Yaskawa INFORM job: A_ROOF_SIDE_0617_2_PAINT_8.JBI

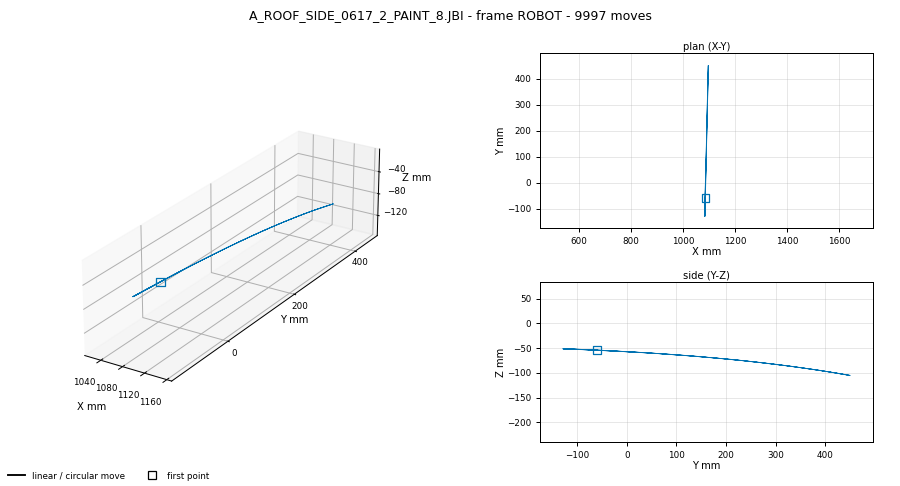
[picture p0: tool path of A_ROOF_SIDE_0617_2_PAINT_8.JBI in frame ROBOT, 9997 of 9997 moves have a stored position in this frame; points joined in program order, loops and branches not executed]
/JOB
//NAME A_ROOF_SIDE_0617_2_PAINT8
//POS
///NPOS 9997,0,0,0,0,0
///TOOL 1
///USER 0
///POSTYPE ROBOT
///RECTAN
///RCONF 1,0,0,0,0,0,0,0,0,0,0,0,0,0,0,0,0,0,0,0,0,0,0,0
C00000=1085.581,-59.825,-53.867,174.286,17.983,152.948
C00001=1085.575,-60.075,-53.857,174.285,17.982,152.948
C00002=1085.569,-60.325,-53.845,174.283,17.980,152.948
C00003=1085.563,-60.574,-53.833,174.282,17.979,152.948
C00004=1085.557,-60.824,-53.822,174.280,17.978,152.948
C00005=1085.551,-61.074,-53.811,174.279,17.976,152.948
C00006=1085.545,-61.323,-53.799,174.277,17.974,152.948
C00007=1085.540,-61.573,-53.788,174.276,17.973,152.948
C00008=1085.534,-61.823,-53.777,174.274,17.972,152.948
C00009=1085.527,-62.072,-53.765,174.273,17.970,152.948
C00010=1085.522,-62.322,-53.754,174.272,17.969,152.948
C00011=1085.515,-62.572,-53.743,174.270,17.968,152.948
C00012=1085.509,-62.821,-53.731,174.269,17.966,152.948
C00013=1085.504,-63.071,-53.719,174.267,17.965,152.948
C00014=1085.498,-63.321,-53.708,174.265,17.963,152.948
C00015=1085.491,-63.571,-53.697,174.264,17.962,152.948
C00016=1085.485,-63.820,-53.685,174.263,17.960,152.948
C00017=1085.480,-64.069,-53.675,174.261,17.959,152.948
C00018=1085.473,-64.320,-53.663,174.260,17.958,152.948
C00019=1085.468,-64.569,-53.651,174.258,17.956,152.948
C00020=1085.461,-64.842,-53.640,174.257,17.955,152.948
C00021=1085.455,-65.116,-53.627,174.254,17.953,152.948
C00022=1085.448,-65.389,-53.615,174.253,17.951,152.948
C00023=1085.442,-65.662,-53.602,174.252,17.950,152.948
C00024=1085.436,-65.912,-53.591,174.250,17.948,152.948
C00025=1085.430,-66.162,-53.580,174.248,17.947,152.948
C00026=1085.424,-66.411,-53.569,174.247,17.946,152.948
C00027=1085.418,-66.661,-53.557,174.246,17.944,152.948
C00028=1085.412,-66.911,-53.546,174.244,17.943,152.948
C00029=1085.407,-67.160,-53.535,174.243,17.942,152.948
C00030=1085.400,-67.410,-53.524,174.241,17.940,152.948
C00031=1085.394,-67.660,-53.513,174.240,17.939,152.948
C00032=1085.389,-67.909,-53.502,174.238,17.937,152.948
C00033=1085.382,-68.159,-53.490,174.237,17.936,152.948
C00034=1085.376,-68.409,-53.479,174.235,17.935,152.948
C00035=1085.371,-68.658,-53.468,174.234,17.933,152.948
C00036=1085.365,-68.909,-53.456,174.232,17.932,152.948
C00037=1085.359,-69.158,-53.445,174.231,17.931,152.948
C00038=1085.354,-69.407,-53.435,174.229,17.929,152.948
C00039=1085.347,-69.658,-53.423,174.228,17.928,152.948
C00040=1085.341,-69.907,-53.412,174.226,17.926,152.948
C00041=1085.336,-70.157,-53.402,174.225,17.925,152.948
C00042=1085.329,-70.406,-53.390,174.223,17.924,152.948
C00043=1085.323,-70.656,-53.379,174.222,17.922,152.948
C00044=1085.318,-70.905,-53.368,174.220,17.921,152.948
C00045=1085.311,-71.155,-53.357,174.219,17.920,152.948
C00046=1085.306,-71.405,-53.346,174.217,17.918,152.948
C00047=1085.300,-71.655,-53.334,174.216,17.917,152.948
C00048=1085.294,-71.905,-53.323,174.214,17.915,152.948
C00049=1085.288,-72.154,-53.312,174.213,17.914,152.948
C00050=1085.283,-72.404,-53.301,174.211,17.913,152.949
C00051=1085.277,-72.653,-53.290,174.210,17.911,152.948
C00052=1085.271,-72.904,-53.279,174.208,17.910,152.948
C00053=1085.265,-73.153,-53.268,174.207,17.909,152.949
C00054=1085.259,-73.403,-53.257,174.205,17.907,152.949
C00055=1085.253,-73.652,-53.246,174.204,17.906,152.949
C00056=1085.247,-73.902,-53.235,174.202,17.904,152.949
C00057=1085.241,-74.152,-53.224,174.201,17.903,152.949
C00058=1085.236,-74.401,-53.213,174.199,17.902,152.949
C00059=1085.229,-74.651,-53.202,174.198,17.900,152.949
C00060=1085.223,-74.901,-53.191,174.196,17.899,152.949
C00061=1085.218,-75.150,-53.180,174.195,17.898,152.949
C00062=1085.211,-75.400,-53.170,174.193,17.896,152.949
C00063=1085.205,-75.650,-53.159,174.192,17.895,152.949
C00064=1085.199,-75.899,-53.148,174.190,17.894,152.949
C00065=1085.193,-76.149,-53.137,174.188,17.893,152.949
C00066=1085.187,-76.399,-53.126,174.187,17.891,152.949
C00067=1085.181,-76.648,-53.115,174.185,17.890,152.949
C00068=1085.176,-76.898,-53.104,174.184,17.889,152.949
C00069=1085.169,-77.148,-53.094,174.182,17.888,152.949
C00070=1085.163,-77.398,-53.083,174.181,17.886,152.949
C00071=1085.157,-77.647,-53.073,174.179,17.885,152.949
C00072=1085.152,-77.897,-53.062,174.178,17.883,152.949
C00073=1085.145,-78.147,-53.050,174.176,17.882,152.949
C00074=1085.140,-78.397,-53.040,174.175,17.881,152.949
C00075=1085.133,-78.646,-53.029,174.174,17.880,152.949
C00076=1085.127,-78.895,-53.018,174.172,17.879,152.949
C00077=1085.121,-79.145,-53.007,174.171,17.878,152.949
C00078=1085.115,-79.395,-52.996,174.169,17.876,152.949
C00079=1085.110,-79.645,-52.986,174.168,17.875,152.949
C00080=1085.104,-79.894,-52.975,174.166,17.874,152.950
C00081=1085.097,-80.144,-52.965,174.165,17.872,152.950
C00082=1085.091,-80.394,-52.954,174.163,17.871,152.950
C00083=1085.086,-80.643,-52.943,174.162,17.870,152.950
C00084=1085.079,-80.920,-52.931,174.160,17.869,152.950
C00085=1085.072,-81.195,-52.919,174.158,17.868,152.950
C00086=1085.065,-81.470,-52.907,174.157,17.866,152.950
C00087=1085.059,-81.746,-52.896,174.154,17.865,152.950
C00088=1085.052,-81.995,-52.886,174.153,17.863,152.950
C00089=1085.046,-82.245,-52.874,174.152,17.862,152.950
C00090=1085.040,-82.495,-52.864,174.150,17.861,152.950
C00091=1085.034,-82.744,-52.854,174.149,17.860,152.950
C00092=1085.028,-82.994,-52.843,174.147,17.859,152.950
C00093=1085.022,-83.244,-52.832,174.146,17.858,152.950
C00094=1085.015,-83.493,-52.822,174.144,17.857,152.950
C00095=1085.010,-83.743,-52.811,174.143,17.855,152.950
C00096=1085.003,-83.993,-52.801,174.141,17.854,152.950
C00097=1084.997,-84.243,-52.790,174.139,17.853,152.951
C00098=1084.991,-84.492,-52.779,174.138,17.851,152.951
C00099=1084.985,-84.742,-52.769,174.136,17.850,152.951
C00100=1084.979,-84.992,-52.759,174.135,17.849,152.951
C00101=1084.972,-85.241,-52.748,174.133,17.848,152.951
C00102=1084.967,-85.492,-52.738,174.132,17.847,152.951
C00103=1084.961,-85.741,-52.727,174.131,17.846,152.951
C00104=1084.955,-85.990,-52.717,174.129,17.845,152.951
C00105=1084.949,-86.240,-52.706,174.128,17.844,152.951
C00106=1084.943,-86.491,-52.695,174.126,17.842,152.951
C00107=1084.936,-86.740,-52.685,174.124,17.841,152.951
C00108=1084.931,-86.990,-52.675,174.123,17.840,152.951
C00109=1084.924,-87.239,-52.665,174.121,17.839,152.951
C00110=1084.919,-87.488,-52.654,174.120,17.838,152.951
C00111=1084.912,-87.739,-52.644,174.118,17.836,152.951
C00112=1084.906,-87.988,-52.633,174.117,17.835,152.952
C00113=1084.900,-88.238,-52.622,174.115,17.834,152.952
C00114=1084.894,-88.488,-52.612,174.114,17.834,152.952
C00115=1084.889,-88.737,-52.602,174.113,17.832,152.952
C00116=1084.882,-88.986,-52.591,174.111,17.831,152.952
C00117=1084.876,-89.237,-52.581,174.109,17.830,152.952
C00118=1084.870,-89.486,-52.570,174.108,17.829,152.952
C00119=1084.864,-89.737,-52.560,174.106,17.827,152.952
C00120=1084.858,-89.986,-52.549,174.105,17.826,152.952
C00121=1084.852,-90.235,-52.539,174.103,17.825,152.952
C00122=1084.847,-90.485,-52.529,174.101,17.824,152.952
C00123=1084.840,-90.734,-52.519,174.101,17.823,152.952
C00124=1084.834,-90.985,-52.508,174.099,17.822,152.952
C00125=1084.828,-91.234,-52.498,174.097,17.821,152.952
C00126=1084.822,-91.485,-52.488,174.096,17.820,152.953
C00127=1084.816,-91.734,-52.477,174.094,17.819,152.953
C00128=1084.810,-91.984,-52.467,174.093,17.817,152.953
C00129=1084.804,-92.233,-52.457,174.091,17.816,152.953
C00130=1084.798,-92.483,-52.446,174.089,17.815,152.953
C00131=1084.793,-92.733,-52.436,174.088,17.814,152.953
C00132=1084.786,-92.982,-52.426,174.087,17.813,152.953
C00133=1084.780,-93.233,-52.415,174.085,17.812,152.953
C00134=1084.774,-93.482,-52.405,174.084,17.811,152.953
C00135=1084.768,-93.732,-52.395,174.082,17.810,152.953
C00136=1084.762,-93.981,-52.384,174.080,17.809,152.953
C00137=1084.756,-94.231,-52.374,174.079,17.807,152.953
C00138=1084.750,-94.480,-52.364,174.077,17.806,152.953
C00139=1084.744,-94.731,-52.354,174.076,17.805,152.954
C00140=1084.738,-94.980,-52.344,174.074,17.804,152.954
C00141=1084.732,-95.230,-52.333,174.073,17.804,152.954
C00142=1084.726,-95.480,-52.324,174.072,17.803,152.954
C00143=1084.720,-95.729,-52.313,174.070,17.801,152.954
C00144=1084.714,-95.979,-52.303,174.068,17.800,152.954
C00145=1084.709,-96.228,-52.292,174.067,17.799,152.954
C00146=1084.702,-96.478,-52.283,174.065,17.798,152.954
C00147=1084.697,-96.728,-52.273,174.063,17.797,152.954
C00148=1084.688,-97.066,-52.259,174.062,17.796,152.954
C00149=1084.680,-97.404,-52.245,174.060,17.794,152.954
C00150=1084.672,-97.741,-52.231,174.058,17.793,152.954
C00151=1084.664,-98.079,-52.218,174.055,17.791,152.955
C00152=1084.658,-98.328,-52.207,174.054,17.790,152.955
C00153=1084.652,-98.578,-52.198,174.053,17.789,152.955
C00154=1084.645,-98.828,-52.188,174.051,17.788,152.955
C00155=1084.640,-99.077,-52.177,174.050,17.787,152.955
C00156=1084.633,-99.328,-52.167,174.048,17.786,152.955
C00157=1084.627,-99.577,-52.158,174.046,17.785,152.955
C00158=1084.621,-99.827,-52.147,174.045,17.784,152.955
C00159=1084.615,-100.077,-52.137,174.044,17.784,152.955
C00160=1084.609,-100.326,-52.128,174.042,17.783,152.956
C00161=1084.603,-100.576,-52.117,174.040,17.782,152.956
C00162=1084.597,-100.826,-52.107,174.039,17.781,152.956
C00163=1084.591,-101.076,-52.098,174.037,17.779,152.956
C00164=1084.584,-101.325,-52.088,174.035,17.778,152.956
C00165=1084.579,-101.575,-52.077,174.035,17.778,152.956
C00166=1084.573,-101.825,-52.068,174.033,17.777,152.956
C00167=1084.566,-102.074,-52.058,174.031,17.776,152.956
C00168=1084.560,-102.324,-52.048,174.030,17.775,152.956
C00169=1084.554,-102.574,-52.038,174.028,17.774,152.957
C00170=1084.548,-102.824,-52.028,174.026,17.773,152.957
C00171=1084.542,-103.073,-52.018,174.026,17.772,152.957
C00172=1084.536,-103.323,-52.008,174.024,17.771,152.957
C00173=1084.530,-103.573,-51.998,174.022,17.770,152.957
C00174=1084.524,-103.822,-51.989,174.021,17.769,152.957
C00175=1084.518,-104.072,-51.978,174.019,17.768,152.957
C00176=1084.512,-104.322,-51.968,174.017,17.767,152.957
C00177=1084.506,-104.571,-51.959,174.016,17.766,152.957
C00178=1084.500,-104.821,-51.949,174.015,17.765,152.957
C00179=1084.493,-105.070,-51.939,174.013,17.764,152.958
C00180=1084.487,-105.320,-51.929,174.011,17.763,152.958
C00181=1084.482,-105.570,-51.919,174.010,17.762,152.958
C00182=1084.475,-105.820,-51.910,174.009,17.762,152.958
C00183=1084.469,-106.070,-51.900,174.007,17.761,152.958
C00184=1084.463,-106.319,-51.890,174.006,17.760,152.958
C00185=1084.457,-106.569,-51.880,174.004,17.758,152.958
C00186=1084.451,-106.819,-51.870,174.002,17.758,152.958
C00187=1084.445,-107.069,-51.860,174.000,17.757,152.959
C00188=1084.439,-107.319,-51.851,173.999,17.756,152.959
C00189=1084.433,-107.568,-51.841,173.998,17.755,152.959
C00190=1084.426,-107.818,-51.831,173.996,17.754,152.959
C00191=1084.420,-108.067,-51.821,173.994,17.753,152.959
C00192=1084.414,-108.317,-51.812,173.993,17.752,152.959
C00193=1084.408,-108.567,-51.802,173.992,17.752,152.959
C00194=1084.402,-108.817,-51.792,173.990,17.751,152.959
C00195=1084.396,-109.067,-51.783,173.988,17.750,152.960
C00196=1084.390,-109.317,-51.773,173.987,17.749,152.960
C00197=1084.384,-109.567,-51.763,173.985,17.748,152.960
C00198=1084.377,-109.816,-51.753,173.984,17.747,152.960
C00199=1084.371,-110.065,-51.744,173.983,17.746,152.960
C00200=1084.365,-110.315,-51.734,173.981,17.746,152.960
C00201=1084.359,-110.565,-51.724,173.979,17.745,152.960
C00202=1084.353,-110.815,-51.715,173.978,17.744,152.960
C00203=1084.347,-111.064,-51.706,173.976,17.743,152.961
C00204=1084.342,-111.284,-51.697,173.975,17.742,152.961
C00205=1084.336,-111.504,-51.688,173.974,17.742,152.961
C00206=1084.331,-111.724,-51.680,173.972,17.741,152.961
C00207=1084.325,-111.944,-51.671,173.970,17.740,152.961
C00208=1084.321,-112.163,-51.663,173.970,17.740,152.961
C00209=1084.315,-112.383,-51.654,173.968,17.739,152.961
C00210=1084.310,-112.604,-51.646,173.967,17.738,152.961
C00211=1084.304,-112.823,-51.638,173.965,17.737,152.962
C00212=1084.298,-113.096,-51.627,173.963,17.736,152.962
C00213=1084.291,-113.370,-51.616,173.962,17.735,152.962
C00214=1084.284,-113.643,-51.606,173.960,17.734,152.962
C00215=1084.277,-113.917,-51.595,173.958,17.734,152.962
C00216=1084.271,-114.167,-51.586,173.957,17.733,152.962
C00217=1084.265,-114.417,-51.576,173.956,17.732,152.962
C00218=1084.259,-114.667,-51.567,173.954,17.731,152.963
C00219=1084.253,-114.916,-51.557,173.952,17.731,152.963
C00220=1084.247,-115.166,-51.548,173.951,17.730,152.963
C00221=1084.241,-115.416,-51.539,173.950,17.729,152.963
C00222=1084.235,-115.666,-51.529,173.948,17.729,152.963
C00223=1084.229,-115.916,-51.520,173.946,17.727,152.963
C00224=1084.223,-116.165,-51.510,173.945,17.727,152.963
C00225=1084.217,-116.415,-51.501,173.943,17.726,152.964
C00226=1084.210,-116.665,-51.491,173.942,17.725,152.964
C00227=1084.203,-116.914,-51.482,173.940,17.724,152.964
C00228=1084.197,-117.164,-51.473,173.939,17.724,152.964
C00229=1084.191,-117.414,-51.463,173.937,17.723,152.964
C00230=1084.186,-117.663,-51.454,173.936,17.722,152.964
C00231=1084.179,-117.913,-51.444,173.934,17.721,152.964
C00232=1084.173,-118.163,-51.435,173.933,17.721,152.965
C00233=1084.167,-118.412,-51.425,173.931,17.720,152.965
C00234=1084.161,-118.663,-51.416,173.929,17.720,152.965
C00235=1084.155,-118.913,-51.407,173.927,17.719,152.965
C00236=1084.149,-119.163,-51.397,173.927,17.718,152.965
C00237=1084.143,-119.412,-51.388,173.925,17.718,152.965
C00238=1084.136,-119.661,-51.379,173.923,17.716,152.966
C00239=1084.130,-119.911,-51.369,173.921,17.715,152.966
C00240=1084.124,-120.161,-51.360,173.920,17.715,152.966
C00241=1084.118,-120.410,-51.350,173.919,17.714,152.966
C00242=1084.112,-120.661,-51.341,173.917,17.714,152.966
C00243=1084.106,-120.911,-51.332,173.915,17.713,152.966
C00244=1084.100,-121.160,-51.323,173.914,17.712,152.966
C00245=1084.094,-121.410,-51.313,173.912,17.712,152.967
C00246=1084.087,-121.659,-51.304,173.911,17.711,152.967
C00247=1084.081,-121.910,-51.295,173.910,17.711,152.967
C00248=1084.075,-122.159,-51.286,173.908,17.710,152.967
C00249=1084.069,-122.409,-51.276,173.906,17.709,152.967
C00250=1084.063,-122.658,-51.267,173.904,17.708,152.968
C00251=1084.057,-122.908,-51.257,173.903,17.708,152.968
C00252=1084.051,-123.158,-51.249,173.901,17.707,152.968
C00253=1084.044,-123.408,-51.240,173.900,17.706,152.968
C00254=1084.038,-123.658,-51.230,173.899,17.706,152.968
C00255=1084.032,-123.907,-51.220,173.897,17.705,152.968
C00256=1084.027,-124.157,-51.211,173.895,17.704,152.969
C00257=1084.020,-124.407,-51.203,173.893,17.703,152.969
C00258=1084.014,-124.656,-51.193,173.892,17.703,152.969
C00259=1084.008,-124.906,-51.184,173.891,17.702,152.969
C00260=1084.002,-125.157,-51.175,173.889,17.702,152.969
C00261=1083.995,-125.405,-51.166,173.888,17.701,152.969
C00262=1083.989,-125.655,-51.157,173.886,17.701,152.970
C00263=1083.983,-125.905,-51.147,173.884,17.700,152.970
C00264=1083.977,-126.156,-51.138,173.882,17.699,152.970
C00265=1083.970,-126.405,-51.129,173.882,17.699,152.970
C00266=1083.965,-126.654,-51.120,173.880,17.698,152.970
C00267=1083.959,-126.905,-51.111,173.878,17.697,152.970
C00268=1083.953,-127.154,-51.102,173.877,17.697,152.971
C00269=1083.946,-127.404,-51.093,173.875,17.696,152.971
C00270=1083.940,-127.654,-51.083,173.873,17.695,152.971
C00271=1083.934,-127.903,-51.075,173.872,17.695,152.971
C00272=1083.928,-128.160,-51.065,173.871,17.694,152.971
C00273=1083.927,-128.416,-51.054,173.869,17.692,152.971
C00274=1083.930,-128.671,-51.042,173.869,17.689,152.971
C00275=1083.937,-128.924,-51.028,173.869,17.684,152.970
C00276=1083.537,-128.945,-51.162,173.825,17.800,153.000
C00277=1083.528,-128.693,-51.176,173.825,17.805,153.001
C00278=1083.525,-128.438,-51.188,173.826,17.808,153.001
C00279=1083.527,-128.182,-51.199,173.827,17.810,153.001
C00280=1083.532,-127.926,-51.209,173.828,17.811,153.001
C00281=1083.538,-127.676,-51.218,173.829,17.812,153.001
C00282=1083.544,-127.426,-51.227,173.831,17.812,153.001
C00283=1083.550,-127.176,-51.237,173.833,17.813,153.001
C00284=1083.556,-126.927,-51.245,173.835,17.814,153.001
C00285=1083.563,-126.677,-51.255,173.836,17.814,153.001
C00286=1083.568,-126.427,-51.264,173.838,17.815,153.000
C00287=1083.575,-126.177,-51.273,173.839,17.816,153.000
C00288=1083.582,-125.927,-51.282,173.840,17.816,153.000
C00289=1083.587,-125.678,-51.291,173.842,17.817,153.000
C00290=1083.593,-125.428,-51.300,173.844,17.817,153.000
C00291=1083.600,-125.178,-51.309,173.846,17.819,152.999
C00292=1083.606,-124.929,-51.319,173.847,17.819,152.999
C00293=1083.612,-124.678,-51.328,173.848,17.820,152.999
C00294=1083.617,-124.429,-51.337,173.850,17.820,152.999
C00295=1083.624,-124.180,-51.346,173.851,17.821,152.999
C00296=1083.631,-123.930,-51.355,173.853,17.821,152.999
C00297=1083.636,-123.679,-51.364,173.855,17.822,152.998
C00298=1083.643,-123.430,-51.374,173.857,17.823,152.998
C00299=1083.649,-123.180,-51.383,173.858,17.823,152.998
C00300=1083.654,-122.931,-51.393,173.859,17.824,152.998
C00301=1083.661,-122.681,-51.401,173.861,17.825,152.998
C00302=1083.667,-122.431,-51.410,173.862,17.825,152.998
C00303=1083.673,-122.181,-51.420,173.864,17.826,152.997
C00304=1083.679,-121.931,-51.429,173.866,17.827,152.997
C00305=1083.685,-121.682,-51.439,173.867,17.828,152.997
C00306=1083.691,-121.432,-51.448,173.868,17.828,152.997
C00307=1083.698,-121.182,-51.457,173.870,17.829,152.997
C00308=1083.704,-120.932,-51.466,173.872,17.829,152.997
C00309=1083.710,-120.683,-51.476,173.874,17.830,152.996
C00310=1083.716,-120.433,-51.485,173.874,17.831,152.996
C00311=1083.722,-120.183,-51.495,173.876,17.832,152.996
C00312=1083.728,-119.933,-51.503,173.878,17.833,152.996
C00313=1083.734,-119.684,-51.513,173.880,17.834,152.996
C00314=1083.741,-119.434,-51.522,173.881,17.834,152.996
C00315=1083.747,-119.184,-51.531,173.882,17.835,152.996
C00316=1083.753,-118.934,-51.541,173.884,17.836,152.995
C00317=1083.759,-118.685,-51.551,173.886,17.836,152.995
C00318=1083.766,-118.435,-51.560,173.887,17.837,152.995
C00319=1083.771,-118.186,-51.569,173.889,17.838,152.995
C00320=1083.777,-117.935,-51.578,173.891,17.838,152.995
C00321=1083.783,-117.686,-51.588,173.892,17.839,152.995
C00322=1083.789,-117.436,-51.597,173.893,17.840,152.995
C00323=1083.795,-117.186,-51.607,173.895,17.840,152.994
C00324=1083.802,-116.936,-51.616,173.897,17.841,152.994
C00325=1083.808,-116.686,-51.626,173.898,17.842,152.994
C00326=1083.815,-116.437,-51.635,173.899,17.842,152.994
C00327=1083.821,-116.187,-51.645,173.901,17.844,152.994
C00328=1083.826,-115.938,-51.654,173.903,17.845,152.994
C00329=1083.833,-115.688,-51.663,173.904,17.846,152.993
C00330=1083.839,-115.438,-51.673,173.905,17.846,152.993
C00331=1083.845,-115.189,-51.682,173.907,17.847,152.993
C00332=1083.851,-114.939,-51.692,173.909,17.848,152.993
C00333=1083.857,-114.689,-51.702,173.910,17.849,152.993
C00334=1083.864,-114.439,-51.711,173.912,17.849,152.993
C00335=1083.870,-114.189,-51.721,173.913,17.850,152.993
C00336=1083.876,-113.940,-51.730,173.915,17.851,152.992
C00337=1083.882,-113.666,-51.740,173.917,17.852,152.992
C00338=1083.888,-113.392,-51.751,173.918,17.853,152.992
C00339=1083.895,-113.118,-51.762,173.920,17.853,152.992
C00340=1083.903,-112.844,-51.772,173.922,17.854,152.992
C00341=1083.909,-112.595,-51.782,173.924,17.856,152.992
C00342=1083.915,-112.345,-51.791,173.924,17.856,152.992
C00343=1083.921,-112.095,-51.801,173.926,17.857,152.992
C00344=1083.927,-111.846,-51.810,173.928,17.858,152.991
C00345=1083.932,-111.596,-51.820,173.930,17.859,152.991
C00346=1083.938,-111.346,-51.830,173.931,17.860,152.991
C00347=1083.944,-111.096,-51.839,173.932,17.860,152.991
C00348=1083.951,-110.846,-51.849,173.934,17.861,152.991
C00349=1083.957,-110.597,-51.859,173.935,17.862,152.991
C00350=1083.963,-110.347,-51.868,173.937,17.863,152.990
C00351=1083.969,-110.097,-51.878,173.939,17.864,152.990
C00352=1083.975,-109.847,-51.887,173.940,17.864,152.990
C00353=1083.982,-109.597,-51.897,173.942,17.865,152.990
C00354=1083.988,-109.348,-51.906,173.943,17.866,152.990
C00355=1083.994,-109.098,-51.917,173.945,17.868,152.990
C00356=1084.000,-108.849,-51.926,173.947,17.869,152.990
C00357=1084.007,-108.599,-51.936,173.948,17.869,152.990
C00358=1084.012,-108.349,-51.946,173.949,17.870,152.990
C00359=1084.018,-108.099,-51.956,173.951,17.871,152.989
C00360=1084.024,-107.849,-51.965,173.953,17.872,152.989
C00361=1084.030,-107.599,-51.975,173.954,17.873,152.989
C00362=1084.037,-107.350,-51.985,173.955,17.873,152.989
C00363=1084.043,-107.100,-51.995,173.957,17.874,152.989
C00364=1084.049,-106.850,-52.004,173.958,17.875,152.989
C00365=1084.055,-106.600,-52.014,173.960,17.876,152.989
C00366=1084.061,-106.351,-52.024,173.962,17.877,152.989
C00367=1084.067,-106.101,-52.033,173.963,17.878,152.989
C00368=1084.074,-105.852,-52.044,173.964,17.879,152.988
C00369=1084.080,-105.602,-52.053,173.966,17.880,152.988
C00370=1084.085,-105.352,-52.063,173.968,17.881,152.988
C00371=1084.091,-105.102,-52.073,173.969,17.882,152.988
C00372=1084.097,-104.852,-52.083,173.971,17.883,152.988
C00373=1084.104,-104.603,-52.093,173.972,17.883,152.988
C00374=1084.109,-104.353,-52.103,173.974,17.884,152.988
C00375=1084.116,-104.103,-52.113,173.975,17.885,152.988
C00376=1084.122,-103.853,-52.122,173.977,17.886,152.987
C00377=1084.128,-103.604,-52.132,173.979,17.887,152.987
C00378=1084.134,-103.354,-52.143,173.980,17.888,152.987
C00379=1084.140,-103.104,-52.152,173.981,17.889,152.987
C00380=1084.146,-102.854,-52.162,173.983,17.890,152.987
C00381=1084.152,-102.605,-52.172,173.984,17.892,152.987
C00382=1084.158,-102.355,-52.182,173.986,17.893,152.987
C00383=1084.164,-102.105,-52.192,173.988,17.894,152.987
C00384=1084.170,-101.855,-52.201,173.989,17.895,152.987
C00385=1084.177,-101.606,-52.212,173.990,17.895,152.987
C00386=1084.182,-101.356,-52.222,173.992,17.896,152.987
C00387=1084.188,-101.106,-52.231,173.993,17.897,152.986
C00388=1084.195,-100.857,-52.242,173.995,17.898,152.986
C00389=1084.200,-100.607,-52.252,173.997,17.899,152.986
C00390=1084.206,-100.357,-52.261,173.998,17.900,152.986
C00391=1084.213,-100.108,-52.272,173.999,17.901,152.986
C00392=1084.219,-99.858,-52.281,174.001,17.902,152.986
C00393=1084.224,-99.608,-52.291,174.003,17.903,152.986
C00394=1084.231,-99.359,-52.302,174.004,17.904,152.986
C00395=1084.237,-99.109,-52.311,174.006,17.905,152.986
C00396=1084.243,-98.859,-52.321,174.008,17.906,152.985
C00397=1084.249,-98.610,-52.332,174.009,17.907,152.985
C00398=1084.255,-98.360,-52.341,174.010,17.908,152.985
C00399=1084.262,-98.110,-52.352,174.012,17.909,152.985
C00400=1084.268,-97.860,-52.362,174.013,17.910,152.985
C00401=1084.275,-97.582,-52.373,174.015,17.911,152.985
C00402=1084.281,-97.304,-52.384,174.017,17.912,152.985
C00403=1084.288,-97.026,-52.395,174.018,17.913,152.985
C00404=1084.295,-96.748,-52.407,174.020,17.914,152.985
C00405=1084.300,-96.498,-52.417,174.021,17.916,152.985
C00406=1084.307,-96.249,-52.428,174.023,17.917,152.985
C00407=1084.313,-95.999,-52.437,174.025,17.918,152.985
C00408=1084.318,-95.750,-52.448,174.026,17.919,152.984
C00409=1084.325,-95.500,-52.458,174.028,17.920,152.984
C00410=1084.330,-95.250,-52.468,174.029,17.922,152.984
C00411=1084.337,-95.001,-52.478,174.031,17.923,152.984
C00412=1084.342,-94.751,-52.488,174.032,17.923,152.984
C00413=1084.348,-94.501,-52.498,174.034,17.924,152.984
C00414=1084.354,-94.251,-52.509,174.035,17.926,152.984
C00415=1084.360,-94.002,-52.519,174.037,17.927,152.984
C00416=1084.366,-93.752,-52.529,174.038,17.928,152.984
C00417=1084.372,-93.503,-52.540,174.040,17.929,152.984
C00418=1084.378,-93.253,-52.550,174.042,17.930,152.984
C00419=1084.384,-93.003,-52.561,174.043,17.932,152.984
C00420=1084.390,-92.753,-52.570,174.044,17.932,152.984
C00421=1084.396,-92.503,-52.581,174.045,17.933,152.984
C00422=1084.402,-92.253,-52.591,174.047,17.934,152.983
C00423=1084.408,-92.004,-52.602,174.049,17.936,152.983
C00424=1084.414,-91.754,-52.611,174.050,17.937,152.983
C00425=1084.420,-91.505,-52.622,174.052,17.938,152.983
C00426=1084.426,-91.255,-52.632,174.054,17.939,152.983
C00427=1084.432,-91.005,-52.643,174.055,17.941,152.983
C00428=1084.439,-90.756,-52.653,174.057,17.942,152.983
C00429=1084.444,-90.505,-52.663,174.058,17.943,152.983
C00430=1084.451,-90.256,-52.674,174.059,17.944,152.983
C00431=1084.456,-90.006,-52.684,174.061,17.945,152.983
C00432=1084.462,-89.757,-52.695,174.062,17.946,152.983
C00433=1084.468,-89.507,-52.705,174.064,17.947,152.983
C00434=1084.474,-89.257,-52.715,174.065,17.948,152.983
C00435=1084.481,-89.007,-52.726,174.067,17.949,152.983
C00436=1084.486,-88.757,-52.736,174.069,17.951,152.982
C00437=1084.493,-88.508,-52.746,174.070,17.952,152.982
C00438=1084.499,-88.259,-52.757,174.072,17.953,152.982
C00439=1084.504,-88.009,-52.767,174.073,17.954,152.982
C00440=1084.510,-87.759,-52.778,174.074,17.955,152.982
C00441=1084.517,-87.509,-52.789,174.076,17.956,152.982
C00442=1084.523,-87.259,-52.798,174.077,17.957,152.982
C00443=1084.529,-87.010,-52.809,174.079,17.959,152.982
C00444=1084.534,-86.760,-52.820,174.080,17.960,152.982
C00445=1084.541,-86.511,-52.830,174.082,17.961,152.982
C00446=1084.547,-86.260,-52.841,174.084,17.962,152.982
C00447=1084.553,-86.011,-52.851,174.085,17.964,152.982
C00448=1084.559,-85.761,-52.861,174.087,17.965,152.982
C00449=1084.565,-85.512,-52.872,174.088,17.966,152.982
C00450=1084.571,-85.262,-52.883,174.090,17.967,152.982
C00451=1084.577,-85.012,-52.893,174.091,17.968,152.982
C00452=1084.584,-84.762,-52.903,174.092,17.969,152.982
C00453=1084.589,-84.513,-52.914,174.094,17.970,152.982
C00454=1084.595,-84.264,-52.925,174.095,17.971,152.981
C00455=1084.602,-84.013,-52.935,174.097,17.973,152.981
C00456=1084.608,-83.764,-52.946,174.098,17.974,152.981
C00457=1084.614,-83.514,-52.956,174.100,17.975,152.981
C00458=1084.620,-83.265,-52.967,174.102,17.977,152.981
C00459=1084.626,-83.014,-52.978,174.103,17.978,152.981
C00460=1084.632,-82.765,-52.988,174.105,17.979,152.981
C00461=1084.638,-82.515,-52.999,174.106,17.980,152.981
C00462=1084.644,-82.266,-53.010,174.108,17.981,152.981
C00463=1084.651,-82.016,-53.020,174.109,17.983,152.981
C00464=1084.656,-81.766,-53.030,174.111,17.984,152.981
C00465=1084.663,-81.491,-53.042,174.113,17.985,152.981
C00466=1084.670,-81.215,-53.054,174.114,17.987,152.981
C00467=1084.677,-80.939,-53.066,174.116,17.988,152.981
C00468=1084.683,-80.663,-53.077,174.117,17.989,152.981
C00469=1084.689,-80.414,-53.088,174.119,17.990,152.981
C00470=1084.696,-80.164,-53.099,174.120,17.991,152.981
C00471=1084.702,-79.915,-53.110,174.122,17.993,152.981
C00472=1084.708,-79.665,-53.121,174.124,17.994,152.980
C00473=1084.714,-79.415,-53.132,174.125,17.995,152.980
C00474=1084.719,-79.165,-53.142,174.127,17.996,152.980
C00475=1084.726,-78.916,-53.152,174.128,17.998,152.980
C00476=1084.732,-78.666,-53.163,174.130,17.999,152.980
C00477=1084.738,-78.416,-53.174,174.131,18.001,152.980
C00478=1084.744,-78.166,-53.185,174.133,18.002,152.980
C00479=1084.749,-77.917,-53.196,174.134,18.003,152.980
C00480=1084.755,-77.667,-53.207,174.136,18.004,152.980
C00481=1084.761,-77.417,-53.218,174.137,18.006,152.980
C00482=1084.768,-77.168,-53.228,174.139,18.007,152.980
C00483=1084.773,-76.918,-53.239,174.140,18.008,152.980
C00484=1084.779,-76.668,-53.250,174.142,18.010,152.980
C00485=1084.785,-76.418,-53.261,174.143,18.011,152.980
C00486=1084.791,-76.169,-53.272,174.145,18.013,152.980
C00487=1084.797,-75.919,-53.283,174.146,18.014,152.980
C00488=1084.803,-75.669,-53.294,174.147,18.015,152.980
C00489=1084.810,-75.420,-53.304,174.149,18.016,152.980
C00490=1084.815,-75.170,-53.315,174.150,18.017,152.980
C00491=1084.822,-74.920,-53.326,174.152,18.018,152.980
C00492=1084.828,-74.671,-53.337,174.153,18.020,152.980
C00493=1084.833,-74.421,-53.348,174.155,18.021,152.980
C00494=1084.839,-74.172,-53.359,174.156,18.023,152.980
C00495=1084.845,-73.922,-53.370,174.158,18.024,152.980
C00496=1084.851,-73.672,-53.381,174.159,18.025,152.980
C00497=1084.857,-73.423,-53.392,174.161,18.027,152.980
C00498=1084.863,-73.172,-53.403,174.162,18.028,152.980
C00499=1084.869,-72.923,-53.414,174.164,18.029,152.980
C00500=1084.875,-72.673,-53.425,174.165,18.031,152.980
C00501=1084.880,-72.424,-53.436,174.167,18.032,152.980
C00502=1084.887,-72.174,-53.447,174.168,18.033,152.980
C00503=1084.892,-71.924,-53.458,174.170,18.035,152.980
C00504=1084.898,-71.675,-53.469,174.171,18.036,152.980
C00505=1084.905,-71.425,-53.480,174.173,18.038,152.980
C00506=1084.910,-71.175,-53.491,174.174,18.039,152.980
C00507=1084.915,-70.925,-53.502,174.176,18.040,152.980
C00508=1084.921,-70.676,-53.514,174.177,18.042,152.980
C00509=1084.928,-70.426,-53.525,174.179,18.043,152.980
C00510=1084.933,-70.177,-53.536,174.180,18.044,152.979
C00511=1084.939,-69.927,-53.547,174.182,18.046,152.980
C00512=1084.946,-69.677,-53.558,174.183,18.048,152.980
C00513=1084.951,-69.428,-53.569,174.184,18.049,152.980
C00514=1084.957,-69.178,-53.580,174.186,18.050,152.979
C00515=1084.963,-68.928,-53.591,174.188,18.052,152.980
C00516=1084.969,-68.678,-53.602,174.189,18.053,152.980
C00517=1084.975,-68.430,-53.614,174.191,18.054,152.979
C00518=1084.981,-68.179,-53.625,174.192,18.056,152.979
C00519=1084.986,-67.930,-53.636,174.193,18.057,152.980
C00520=1084.992,-67.680,-53.647,174.195,18.059,152.979
C00521=1084.999,-67.430,-53.658,174.197,18.060,152.979
C00522=1085.004,-67.180,-53.669,174.198,18.062,152.979
C00523=1085.010,-66.932,-53.681,174.199,18.063,152.980
C00524=1085.017,-66.681,-53.692,174.201,18.064,152.979
C00525=1085.022,-66.432,-53.703,174.202,18.066,152.979
C00526=1085.028,-66.181,-53.715,174.204,18.067,152.979
C00527=1085.034,-65.932,-53.726,174.205,18.068,152.979
C00528=1085.040,-65.683,-53.737,174.207,18.070,152.979
C00529=1085.046,-65.409,-53.750,174.209,18.072,152.979
C00530=1085.053,-65.135,-53.762,174.211,18.074,152.979
C00531=1085.059,-64.861,-53.774,174.212,18.075,152.979
C00532=1085.066,-64.588,-53.786,174.214,18.076,152.979
C00533=1085.072,-64.339,-53.798,174.215,18.078,152.979
C00534=1085.078,-64.089,-53.809,174.216,18.079,152.979
C00535=1085.084,-63.839,-53.820,174.218,18.081,152.979
C00536=1085.089,-63.590,-53.831,174.219,18.082,152.979
C00537=1085.096,-63.340,-53.843,174.221,18.084,152.979
C00538=1085.102,-63.091,-53.854,174.222,18.085,152.979
C00539=1085.107,-62.840,-53.866,174.225,18.087,152.979
C00540=1085.114,-62.591,-53.877,174.226,18.088,152.979
C00541=1085.120,-62.341,-53.889,174.228,18.090,152.979
C00542=1085.126,-62.092,-53.900,174.229,18.091,152.979
C00543=1085.132,-61.843,-53.911,174.230,18.093,152.979
C00544=1085.137,-61.592,-53.923,174.232,18.094,152.979
C00545=1085.143,-61.343,-53.934,174.233,18.096,152.979
C00546=1085.150,-61.093,-53.946,174.235,18.097,152.979
C00547=1085.155,-60.844,-53.957,174.236,18.099,152.979
C00548=1085.162,-60.594,-53.968,174.238,18.100,152.979
C00549=1085.167,-60.344,-53.980,174.239,18.101,152.979
C00550=1085.173,-60.094,-53.991,174.241,18.103,152.979
C00551=1085.179,-59.845,-54.002,174.242,18.104,152.979
C00552=1085.186,-59.595,-54.014,174.244,18.105,152.979
C00553=1085.191,-59.346,-54.025,174.245,18.107,152.979
C00554=1085.197,-59.096,-54.038,174.247,18.109,152.979
C00555=1085.203,-58.846,-54.049,174.248,18.110,152.979
C00556=1085.209,-58.596,-54.060,174.249,18.112,152.979
C00557=1085.216,-58.347,-54.071,174.251,18.113,152.979
C00558=1085.221,-58.097,-54.083,174.253,18.114,152.979
C00559=1085.227,-57.848,-54.095,174.254,18.116,152.979
C00560=1085.233,-57.598,-54.106,174.255,18.117,152.979
C00561=1085.240,-57.349,-54.118,174.257,18.119,152.980
C00562=1085.246,-57.099,-54.129,174.259,18.120,152.979
C00563=1085.251,-56.849,-54.140,174.261,18.122,152.979
C00564=1085.258,-56.599,-54.152,174.262,18.124,152.979
C00565=1085.263,-56.350,-54.163,174.264,18.125,152.979
C00566=1085.269,-56.100,-54.176,174.265,18.127,152.980
C00567=1085.276,-55.850,-54.187,174.267,18.128,152.979
C00568=1085.282,-55.601,-54.199,174.268,18.129,152.979
C00569=1085.288,-55.351,-54.210,174.269,18.131,152.979
C00570=1085.293,-55.101,-54.222,174.271,18.132,152.980
C00571=1085.300,-54.851,-54.233,174.272,18.134,152.980
C00572=1085.306,-54.602,-54.245,174.274,18.135,152.979
C00573=1085.312,-54.352,-54.256,174.275,18.137,152.979
C00574=1085.318,-54.102,-54.269,174.277,18.138,152.980
C00575=1085.324,-53.853,-54.280,174.278,18.140,152.980
C00576=1085.330,-53.603,-54.291,174.280,18.141,152.980
C00577=1085.336,-53.354,-54.304,174.281,18.142,152.979
C00578=1085.342,-53.104,-54.315,174.283,18.144,152.979
C00579=1085.349,-52.854,-54.327,174.285,18.146,152.980
C00580=1085.354,-52.605,-54.338,174.286,18.148,152.980
C00581=1085.360,-52.355,-54.350,174.288,18.149,152.980
C00582=1085.366,-52.106,-54.362,174.289,18.151,152.980
C00583=1085.373,-51.856,-54.373,174.291,18.152,152.980
C00584=1085.378,-51.606,-54.386,174.292,18.153,152.980
C00585=1085.384,-51.356,-54.397,174.294,18.155,152.980
C00586=1085.391,-51.107,-54.409,174.295,18.156,152.980
C00587=1085.397,-50.857,-54.421,174.296,18.158,152.980
C00588=1085.402,-50.607,-54.432,174.298,18.160,152.980
C00589=1085.409,-50.358,-54.444,174.299,18.161,152.980
C00590=1085.414,-50.108,-54.455,174.301,18.162,152.980
C00591=1085.421,-49.859,-54.467,174.303,18.164,152.980
C00592=1085.426,-49.609,-54.480,174.304,18.166,152.980
C00593=1085.433,-49.336,-54.492,174.306,18.167,152.980
C00594=1085.439,-49.065,-54.506,174.307,18.169,152.980
C00595=1085.445,-48.792,-54.518,174.310,18.171,152.980
C00596=1085.452,-48.520,-54.532,174.311,18.173,152.980
C00597=1085.458,-48.271,-54.543,174.312,18.174,152.980
C00598=1085.464,-48.021,-54.555,174.314,18.176,152.980
C00599=1085.470,-47.772,-54.567,174.315,18.177,152.980
C00600=1085.475,-47.521,-54.579,174.317,18.179,152.980
C00601=1085.482,-47.272,-54.591,174.318,18.180,152.980
C00602=1085.487,-47.023,-54.603,174.319,18.182,152.980
C00603=1085.493,-46.773,-54.616,174.321,18.183,152.980
C00604=1085.499,-46.523,-54.626,174.323,18.186,152.980
C00605=1085.505,-46.273,-54.639,174.324,18.187,152.980
C00606=1085.511,-46.024,-54.651,174.326,18.189,152.980
C00607=1085.517,-45.775,-54.663,174.327,18.190,152.980
C00608=1085.522,-45.524,-54.675,174.329,18.192,152.980
C00609=1085.532,-45.122,-54.694,174.331,18.194,152.980
C00610=1085.541,-44.720,-54.714,174.334,18.197,152.980
C00611=1085.551,-44.318,-54.733,174.336,18.200,152.980
C00612=1085.560,-43.916,-54.753,174.339,18.203,152.980
C00613=1085.567,-43.666,-54.765,174.340,18.204,152.981
C00614=1085.573,-43.416,-54.777,174.341,18.206,152.981
C00615=1085.579,-43.167,-54.788,174.343,18.207,152.981
C00616=1085.584,-42.917,-54.801,174.344,18.209,152.981
C00617=1085.590,-42.667,-54.813,174.346,18.210,152.981
C00618=1085.596,-42.418,-54.825,174.347,18.212,152.981
C00619=1085.602,-42.168,-54.837,174.348,18.214,152.981
C00620=1085.608,-41.918,-54.850,174.351,18.216,152.981
C00621=1085.615,-41.669,-54.862,174.352,18.217,152.981
C00622=1085.620,-41.419,-54.873,174.353,18.219,152.981
C00623=1085.626,-41.169,-54.886,174.355,18.220,152.981
C00624=1085.632,-40.920,-54.898,174.356,18.222,152.981
C00625=1085.638,-40.670,-54.910,174.358,18.223,152.981
C00626=1085.644,-40.420,-54.923,174.359,18.225,152.981
C00627=1085.650,-40.171,-54.934,174.361,18.227,152.981
C00628=1085.656,-39.922,-54.947,174.363,18.229,152.981
C00629=1085.662,-39.672,-54.959,174.364,18.230,152.981
C00630=1085.668,-39.422,-54.971,174.366,18.232,152.981
C00631=1085.674,-39.172,-54.984,174.367,18.233,152.981
C00632=1085.679,-38.923,-54.996,174.368,18.235,152.981
C00633=1085.686,-38.674,-55.008,174.370,18.236,152.981
C00634=1085.692,-38.424,-55.020,174.371,18.238,152.981
C00635=1085.698,-38.173,-55.032,174.373,18.240,152.981
C00636=1085.703,-37.924,-55.044,174.375,18.242,152.981
C00637=1085.709,-37.674,-55.057,174.376,18.243,152.981
C00638=1085.715,-37.425,-55.069,174.378,18.245,152.981
C00639=1085.721,-37.175,-55.081,174.379,18.246,152.981
C00640=1085.727,-36.926,-55.094,174.381,18.248,152.981
C00641=1085.733,-36.676,-55.106,174.382,18.249,152.981
C00642=1085.738,-36.426,-55.118,174.383,18.251,152.982
C00643=1085.744,-36.177,-55.131,174.385,18.254,152.982
C00644=1085.750,-35.927,-55.143,174.387,18.255,152.982
C00645=1085.757,-35.678,-55.156,174.388,18.257,152.982
C00646=1085.762,-35.429,-55.168,174.390,18.258,152.982
C00647=1085.768,-35.179,-55.181,174.391,18.260,152.982
C00648=1085.774,-34.929,-55.194,174.392,18.261,152.982
C00649=1085.780,-34.679,-55.206,174.394,18.263,152.982
C00650=1085.785,-34.430,-55.218,174.396,18.265,152.982
C00651=1085.791,-34.180,-55.231,174.397,18.267,152.982
C00652=1085.797,-33.930,-55.243,174.399,18.269,152.982
C00653=1085.806,-33.561,-55.261,174.401,18.271,152.982
C00654=1085.815,-33.193,-55.280,174.403,18.273,152.982
C00655=1085.823,-32.824,-55.298,174.405,18.275,152.982
C00656=1085.832,-32.455,-55.317,174.408,18.278,152.982
C00657=1085.838,-32.205,-55.329,174.409,18.280,152.982
C00658=1085.844,-31.956,-55.341,174.411,18.282,152.982
C00659=1085.849,-31.706,-55.354,174.412,18.283,152.982
C00660=1085.855,-31.456,-55.367,174.413,18.285,152.983
C00661=1085.861,-31.206,-55.379,174.415,18.287,152.983
C00662=1085.868,-30.957,-55.392,174.417,18.289,152.983
C00663=1085.873,-30.708,-55.405,174.418,18.290,152.983
C00664=1085.879,-30.458,-55.417,174.420,18.292,152.983
C00665=1085.885,-30.208,-55.430,174.421,18.294,152.983
C00666=1085.891,-29.958,-55.442,174.423,18.295,152.983
C00667=1085.897,-29.709,-55.456,174.424,18.297,152.983
C00668=1085.903,-29.459,-55.468,174.426,18.299,152.983
C00669=1085.909,-29.210,-55.480,174.427,18.301,152.983
C00670=1085.915,-28.960,-55.492,174.429,18.302,152.983
C00671=1085.921,-28.711,-55.506,174.430,18.304,152.983
C00672=1085.927,-28.461,-55.518,174.432,18.305,152.983
C00673=1085.933,-28.211,-55.531,174.433,18.307,152.983
C00674=1085.939,-27.961,-55.543,174.435,18.309,152.983
C00675=1085.945,-27.712,-55.556,174.437,18.311,152.983
C00676=1085.950,-27.463,-55.569,174.438,18.312,152.983
C00677=1085.956,-27.213,-55.581,174.440,18.314,152.983
C00678=1085.962,-26.963,-55.594,174.441,18.316,152.983
C00679=1085.968,-26.714,-55.607,174.442,18.317,152.984
C00680=1085.974,-26.464,-55.620,174.444,18.319,152.984
C00681=1085.980,-26.214,-55.632,174.446,18.321,152.984
C00682=1085.986,-25.965,-55.645,174.447,18.323,152.984
C00683=1085.991,-25.715,-55.658,174.448,18.325,152.984
C00684=1085.997,-25.466,-55.671,174.450,18.326,152.984
C00685=1086.003,-25.216,-55.684,174.452,18.328,152.984
C00686=1086.009,-24.966,-55.697,174.453,18.330,152.984
C00687=1086.015,-24.717,-55.709,174.455,18.331,152.984
C00688=1086.021,-24.467,-55.722,174.456,18.333,152.984
C00689=1086.026,-24.218,-55.735,174.457,18.335,152.984
C00690=1086.031,-23.968,-55.748,174.459,18.337,152.984
C00691=1086.038,-23.719,-55.761,174.461,18.339,152.984
C00692=1086.043,-23.469,-55.774,174.463,18.340,152.984
C00693=1086.049,-23.219,-55.786,174.464,18.342,152.984
C00694=1086.056,-22.970,-55.799,174.465,18.344,152.984
C00695=1086.062,-22.720,-55.812,174.467,18.345,152.984
C00696=1086.068,-22.470,-55.825,174.469,18.347,152.984
C00697=1086.072,-22.221,-55.838,174.470,18.349,152.985
C00698=1086.079,-21.972,-55.851,174.471,18.351,152.985
C00699=1086.084,-21.722,-55.864,174.473,18.353,152.985
C00700=1086.090,-21.472,-55.876,174.474,18.354,152.985
C00701=1086.097,-21.223,-55.890,174.476,18.356,152.985
C00702=1086.102,-20.972,-55.903,174.478,18.358,152.985
C00703=1086.108,-20.723,-55.916,174.479,18.360,152.985
C00704=1086.114,-20.473,-55.929,174.480,18.361,152.985
C00705=1086.120,-20.224,-55.942,174.482,18.363,152.985
C00706=1086.126,-19.974,-55.954,174.484,18.365,152.985
C00707=1086.131,-19.725,-55.968,174.485,18.367,152.985
C00708=1086.137,-19.475,-55.981,174.487,18.369,152.985
C00709=1086.144,-19.225,-55.994,174.488,18.370,152.985
C00710=1086.149,-18.976,-56.006,174.489,18.372,152.985
C00711=1086.155,-18.727,-56.020,174.492,18.374,152.985
C00712=1086.160,-18.477,-56.033,174.493,18.375,152.985
C00713=1086.166,-18.228,-56.046,174.494,18.377,152.986
C00714=1086.172,-17.978,-56.059,174.496,18.379,152.986
C00715=1086.179,-17.728,-56.072,174.497,18.381,152.986
C00716=1086.185,-17.479,-56.085,174.499,18.383,152.986
C00717=1086.191,-17.206,-56.099,174.501,18.384,152.986
C00718=1086.198,-16.933,-56.114,174.502,18.386,152.986
C00719=1086.204,-16.660,-56.128,174.504,18.388,152.986
C00720=1086.210,-16.388,-56.142,174.506,18.390,152.986
C00721=1086.216,-16.138,-56.156,174.508,18.392,152.986
C00722=1086.222,-15.889,-56.168,174.509,18.394,152.986
C00723=1086.228,-15.639,-56.182,174.510,18.396,152.986
C00724=1086.234,-15.390,-56.195,174.512,18.397,152.986
C00725=1086.240,-15.140,-56.208,174.513,18.399,152.986
C00726=1086.246,-14.891,-56.221,174.515,18.401,152.986
C00727=1086.251,-14.640,-56.234,174.517,18.403,152.986
C00728=1086.257,-14.391,-56.248,174.518,18.404,152.986
C00729=1086.263,-14.142,-56.261,174.520,18.406,152.987
C00730=1086.269,-13.892,-56.274,174.521,18.408,152.987
C00731=1086.274,-13.642,-56.288,174.523,18.410,152.987
C00732=1086.280,-13.393,-56.301,174.524,18.412,152.987
C00733=1086.286,-13.143,-56.314,174.526,18.413,152.987
C00734=1086.292,-12.893,-56.328,174.527,18.415,152.987
C00735=1086.298,-12.644,-56.341,174.529,18.417,152.987
C00736=1086.304,-12.395,-56.355,174.531,18.419,152.987
C00737=1086.309,-12.145,-56.367,174.532,18.420,152.987
C00738=1086.315,-11.895,-56.381,174.533,18.422,152.987
C00739=1086.321,-11.646,-56.394,174.535,18.425,152.987
C00740=1086.327,-11.396,-56.407,174.537,18.426,152.987
C00741=1086.333,-11.146,-56.421,174.538,18.428,152.987
C00742=1086.339,-10.897,-56.434,174.539,18.430,152.988
C00743=1086.344,-10.648,-56.448,174.541,18.431,152.988
C00744=1086.350,-10.398,-56.461,174.543,18.433,152.988
C00745=1086.356,-10.148,-56.474,174.544,18.435,152.988
C00746=1086.362,-9.899,-56.488,174.546,18.437,152.988
C00747=1086.367,-9.649,-56.502,174.547,18.438,152.988
C00748=1086.374,-9.400,-56.515,174.549,18.441,152.988
C00749=1086.379,-9.150,-56.528,174.550,18.443,152.988
C00750=1086.385,-8.901,-56.541,174.552,18.444,152.988
C00751=1086.390,-8.651,-56.555,174.553,18.446,152.988
C00752=1086.397,-8.402,-56.568,174.556,18.448,152.988
C00753=1086.402,-8.152,-56.582,174.557,18.450,152.988
C00754=1086.409,-7.902,-56.596,174.558,18.451,152.988
C00755=1086.414,-7.652,-56.609,174.560,18.453,152.988
C00756=1086.420,-7.403,-56.622,174.562,18.455,152.988
C00757=1086.426,-7.153,-56.636,174.563,18.457,152.989
C00758=1086.432,-6.904,-56.649,174.564,18.459,152.989
C00759=1086.437,-6.654,-56.663,174.566,18.460,152.989
C00760=1086.444,-6.405,-56.677,174.567,18.462,152.989
C00761=1086.449,-6.155,-56.690,174.569,18.464,152.989
C00762=1086.455,-5.906,-56.704,174.571,18.466,152.989
C00763=1086.461,-5.655,-56.717,174.572,18.467,152.989
C00764=1086.467,-5.406,-56.730,174.573,18.469,152.989
C00765=1086.473,-5.156,-56.744,174.576,18.471,152.989
C00766=1086.479,-4.907,-56.758,174.577,18.473,152.989
C00767=1086.485,-4.658,-56.771,174.578,18.475,152.989
C00768=1086.491,-4.408,-56.785,174.580,18.476,152.989
C00769=1086.496,-4.159,-56.799,174.582,18.478,152.989
C00770=1086.502,-3.909,-56.812,174.583,18.480,152.989
C00771=1086.508,-3.659,-56.826,174.585,18.482,152.989
C00772=1086.515,-3.410,-56.839,174.586,18.483,152.990
C00773=1086.520,-3.160,-56.853,174.588,18.485,152.989
C00774=1086.526,-2.911,-56.867,174.589,18.488,152.990
C00775=1086.531,-2.661,-56.881,174.591,18.489,152.990
C00776=1086.537,-2.412,-56.894,174.593,18.491,152.990
C00777=1086.543,-2.162,-56.908,174.594,18.493,152.990
C00778=1086.548,-1.913,-56.922,174.596,18.495,152.990
C00779=1086.554,-1.663,-56.936,174.597,18.496,152.990
C00780=1086.561,-1.413,-56.949,174.599,18.499,152.990
C00781=1086.567,-1.140,-56.965,174.601,18.500,152.990
C00782=1086.573,-0.865,-56.980,174.603,18.503,152.990
C00783=1086.579,-0.591,-56.995,174.604,18.505,152.990
C00784=1086.586,-0.316,-57.010,174.606,18.507,152.991
C00785=1086.591,-0.067,-57.024,174.607,18.509,152.991
C00786=1086.597,0.183,-57.038,174.609,18.510,152.991
C00787=1086.602,0.432,-57.052,174.610,18.512,152.991
C00788=1086.608,0.682,-57.065,174.612,18.514,152.991
C00789=1086.614,0.932,-57.079,174.614,18.516,152.991
C00790=1086.620,1.181,-57.093,174.615,18.517,152.991
C00791=1086.625,1.431,-57.107,174.616,18.520,152.991
C00792=1086.631,1.680,-57.122,174.618,18.522,152.991
C00793=1086.637,1.929,-57.135,174.620,18.523,152.991
C00794=1086.643,2.179,-57.149,174.621,18.525,152.991
C00795=1086.649,2.429,-57.163,174.622,18.527,152.991
C00796=1086.654,2.679,-57.177,174.625,18.529,152.991
C00797=1086.660,2.928,-57.191,174.626,18.531,152.992
C00798=1086.666,3.177,-57.204,174.627,18.532,152.992
C00799=1086.672,3.426,-57.219,174.630,18.535,152.992
C00800=1086.677,3.676,-57.232,174.631,18.536,152.992
C00801=1086.683,3.926,-57.247,174.632,18.538,152.992
C00802=1086.689,4.176,-57.261,174.634,18.540,152.992
C00803=1086.694,4.425,-57.274,174.636,18.542,152.992
C00804=1086.701,4.674,-57.288,174.637,18.544,152.992
C00805=1086.707,4.924,-57.303,174.638,18.545,152.992
C00806=1086.712,5.174,-57.317,174.641,18.547,152.992
C00807=1086.718,5.424,-57.330,174.642,18.549,152.992
C00808=1086.724,5.672,-57.345,174.643,18.551,152.992
C00809=1086.729,5.922,-57.359,174.645,18.553,152.992
C00810=1086.735,6.172,-57.373,174.647,18.555,152.992
C00811=1086.741,6.422,-57.386,174.648,18.557,152.993
C00812=1086.747,6.671,-57.401,174.650,18.558,152.993
C00813=1086.753,6.920,-57.415,174.652,18.560,152.993
C00814=1086.759,7.170,-57.429,174.653,18.562,152.993
C00815=1086.764,7.420,-57.443,174.654,18.564,152.993
C00816=1086.770,7.669,-57.457,174.656,18.565,152.993
C00817=1086.776,7.919,-57.472,174.658,18.568,152.993
C00818=1086.782,8.169,-57.486,174.659,18.569,152.993
C00819=1086.788,8.417,-57.500,174.661,18.571,152.993
C00820=1086.794,8.667,-57.513,174.663,18.573,152.993
C00821=1086.800,8.917,-57.528,174.664,18.575,152.993
C00822=1086.805,9.166,-57.542,174.665,18.577,152.993
C00823=1086.811,9.416,-57.556,174.667,18.578,152.993
C00824=1086.817,9.665,-57.571,174.669,18.580,152.993
C00825=1086.823,9.915,-57.585,174.671,18.582,152.993
C00826=1086.828,10.165,-57.599,174.672,18.584,152.994
C00827=1086.835,10.414,-57.614,174.674,18.586,152.994
C00828=1086.840,10.664,-57.628,174.675,18.588,152.994
C00829=1086.846,10.913,-57.641,174.677,18.589,152.994
C00830=1086.853,11.163,-57.656,174.679,18.591,152.994
C00831=1086.858,11.412,-57.670,174.680,18.593,152.994
C00832=1086.864,11.661,-57.684,174.682,18.595,152.994
C00833=1086.870,11.912,-57.698,174.683,18.596,152.994
C00834=1086.876,12.161,-57.713,174.685,18.598,152.994
C00835=1086.881,12.410,-57.727,174.687,18.600,152.994
C00836=1086.888,12.660,-57.742,174.688,18.602,152.994
C00837=1086.893,12.909,-57.756,174.690,18.604,152.994
C00838=1086.899,13.158,-57.770,174.692,18.606,152.994
C00839=1086.905,13.409,-57.785,174.693,18.608,152.994
C00840=1086.911,13.658,-57.799,174.695,18.610,152.994
C00841=1086.917,13.908,-57.813,174.697,18.611,152.994
C00842=1086.923,14.157,-57.828,174.698,18.613,152.995
C00843=1086.928,14.406,-57.842,174.699,18.614,152.995
C00844=1086.934,14.656,-57.857,174.701,18.617,152.995
C00845=1086.941,14.932,-57.873,174.703,18.619,152.995
C00846=1086.947,15.208,-57.888,174.705,18.621,152.995
C00847=1086.954,15.485,-57.905,174.706,18.623,152.995
C00848=1086.960,15.761,-57.920,174.708,18.625,152.995
C00849=1086.965,16.011,-57.934,174.710,18.627,152.995
C00850=1086.972,16.260,-57.949,174.712,18.629,152.995
C00851=1086.977,16.510,-57.963,174.713,18.630,152.995
C00852=1086.982,16.759,-57.978,174.715,18.632,152.995
C00853=1086.989,17.009,-57.993,174.717,18.634,152.995
C00854=1086.994,17.258,-58.007,174.718,18.636,152.995
C00855=1087.000,17.508,-58.022,174.720,18.638,152.995
C00856=1087.006,17.757,-58.036,174.722,18.640,152.996
C00857=1087.012,18.006,-58.050,174.723,18.642,152.996
C00858=1087.018,18.256,-58.065,174.724,18.643,152.996
C00859=1087.023,18.506,-58.080,174.726,18.645,152.996
C00860=1087.029,18.756,-58.095,174.728,18.647,152.996
C00861=1087.035,19.005,-58.109,174.729,18.649,152.996
C00862=1087.040,19.254,-58.123,174.731,18.650,152.996
C00863=1087.047,19.504,-58.138,174.733,18.652,152.996
C00864=1087.053,19.753,-58.153,174.734,18.655,152.996
C00865=1087.058,20.003,-58.168,174.736,18.656,152.996
C00866=1087.064,20.252,-58.182,174.738,18.658,152.996
C00867=1087.070,20.501,-58.197,174.739,18.660,152.996
C00868=1087.076,20.752,-58.211,174.740,18.662,152.996
C00869=1087.081,21.001,-58.226,174.743,18.664,152.996
C00870=1087.087,21.250,-58.241,174.744,18.665,152.996
C00871=1087.093,21.499,-58.256,174.746,18.667,152.997
C00872=1087.098,21.750,-58.270,174.748,18.669,152.997
C00873=1087.104,21.999,-58.285,174.749,18.671,152.997
C00874=1087.110,22.248,-58.300,174.750,18.673,152.997
C00875=1087.116,22.498,-58.315,174.753,18.675,152.997
C00876=1087.121,22.747,-58.329,174.754,18.677,152.997
C00877=1087.127,22.997,-58.344,174.755,18.678,152.997
C00878=1087.133,23.246,-58.359,174.758,18.680,152.997
C00879=1087.139,23.496,-58.374,174.759,18.682,152.997
C00880=1087.144,23.745,-58.389,174.760,18.684,152.997
C00881=1087.151,23.995,-58.403,174.762,18.686,152.997
C00882=1087.156,24.245,-58.418,174.764,18.687,152.997
C00883=1087.162,24.494,-58.433,174.765,18.689,152.997
C00884=1087.168,24.743,-58.448,174.767,18.692,152.997
C00885=1087.174,24.992,-58.462,174.769,18.693,152.998
C00886=1087.179,25.242,-58.478,174.770,18.695,152.998
C00887=1087.185,25.492,-58.492,174.772,18.697,152.998
C00888=1087.191,25.741,-58.507,174.774,18.698,152.998
C00889=1087.196,25.991,-58.522,174.776,18.701,152.998
C00890=1087.202,26.240,-58.537,174.777,18.702,152.998
C00891=1087.208,26.490,-58.552,174.779,18.704,152.998
C00892=1087.214,26.739,-58.567,174.781,18.706,152.998
C00893=1087.220,26.988,-58.581,174.782,18.707,152.998
C00894=1087.225,27.238,-58.597,174.784,18.710,152.998
C00895=1087.232,27.488,-58.612,174.786,18.712,152.998
C00896=1087.237,27.737,-58.626,174.787,18.713,152.998
C00897=1087.243,27.987,-58.641,174.789,18.715,152.998
C00898=1087.249,28.236,-58.656,174.791,18.717,152.998
C00899=1087.254,28.486,-58.671,174.792,18.719,152.998
C00900=1087.260,28.735,-58.686,174.794,18.720,152.998
C00901=1087.266,28.985,-58.701,174.796,18.722,152.998
C00902=1087.271,29.234,-58.716,174.797,18.724,152.998
C00903=1087.277,29.484,-58.732,174.798,18.726,152.999
C00904=1087.283,29.733,-58.746,174.801,18.728,152.999
C00905=1087.289,29.983,-58.762,174.802,18.730,152.999
C00906=1087.294,30.232,-58.776,174.804,18.732,152.999
C00907=1087.300,30.482,-58.792,174.806,18.734,152.999
C00908=1087.306,30.731,-58.806,174.807,18.735,152.999
C00909=1087.312,31.009,-58.824,174.809,18.737,152.999
C00910=1087.319,31.286,-58.841,174.811,18.740,152.999
C00911=1087.325,31.564,-58.858,174.813,18.741,152.999
C00912=1087.331,31.842,-58.874,174.815,18.743,152.999
C00913=1087.336,32.091,-58.889,174.816,18.745,152.999
C00914=1087.343,32.341,-58.904,174.818,18.748,152.999
C00915=1087.349,32.590,-58.920,174.820,18.749,152.999
C00916=1087.355,32.839,-58.935,174.821,18.751,152.999
C00917=1087.360,33.089,-58.950,174.824,18.753,152.999
C00918=1087.366,33.338,-58.965,174.825,18.754,152.999
C00919=1087.372,33.588,-58.981,174.826,18.756,153.000
C00920=1087.377,33.837,-58.995,174.828,18.758,153.000
C00921=1087.383,34.087,-59.011,174.830,18.760,153.000
C00922=1087.389,34.337,-59.026,174.831,18.761,153.000
C00923=1087.395,34.586,-59.041,174.834,18.763,153.000
C00924=1087.400,34.835,-59.057,174.835,18.766,153.000
C00925=1087.406,35.084,-59.072,174.837,18.768,153.000
C00926=1087.412,35.334,-59.087,174.838,18.769,153.000
C00927=1087.418,35.584,-59.102,174.840,18.771,153.000
C00928=1087.423,35.833,-59.117,174.842,18.773,153.000
C00929=1087.429,36.082,-59.134,174.843,18.774,153.000
C00930=1087.436,36.332,-59.149,174.845,18.776,153.000
C00931=1087.441,36.581,-59.164,174.847,18.778,153.000
C00932=1087.447,36.831,-59.179,174.848,18.780,153.000
C00933=1087.453,37.081,-59.194,174.851,18.782,153.000
C00934=1087.458,37.330,-59.210,174.852,18.783,153.000
C00935=1087.464,37.579,-59.225,174.853,18.785,153.000
C00936=1087.470,37.829,-59.241,174.856,18.787,153.000
C00937=1087.475,38.079,-59.256,174.857,18.789,153.001
C00938=1087.482,38.328,-59.271,174.859,18.791,153.001
C00939=1087.487,38.577,-59.287,174.861,18.793,153.001
C00940=1087.493,38.827,-59.302,174.862,18.794,153.001
C00941=1087.498,39.077,-59.318,174.864,18.796,153.001
C00942=1087.504,39.325,-59.333,174.866,18.798,153.001
C00943=1087.510,39.575,-59.349,174.868,18.800,153.001
C00944=1087.516,39.825,-59.364,174.869,18.802,153.001
C00945=1087.521,40.074,-59.380,174.871,18.804,153.001
C00946=1087.527,40.324,-59.395,174.873,18.806,153.001
C00947=1087.533,40.573,-59.410,174.874,18.807,153.001
C00948=1087.538,40.822,-59.426,174.877,18.809,153.001
C00949=1087.544,41.072,-59.442,174.878,18.811,153.001
C00950=1087.550,41.322,-59.457,174.879,18.813,153.001
C00951=1087.556,41.570,-59.473,174.881,18.815,153.001
C00952=1087.561,41.820,-59.488,174.883,18.816,153.001
C00953=1087.567,42.070,-59.504,174.884,18.818,153.001
C00954=1087.572,42.319,-59.520,174.887,18.820,153.001
C00955=1087.578,42.569,-59.535,174.888,18.821,153.001
C00956=1087.585,42.818,-59.551,174.890,18.824,153.002
C00957=1087.590,43.067,-59.566,174.891,18.826,153.002
C00958=1087.596,43.316,-59.582,174.894,18.828,153.002
C00959=1087.601,43.566,-59.598,174.895,18.829,153.002
C00960=1087.607,43.816,-59.613,174.897,18.831,153.002
C00961=1087.612,44.065,-59.629,174.899,18.833,153.002
C00962=1087.618,44.315,-59.645,174.900,18.834,153.002
C00963=1087.624,44.564,-59.661,174.902,18.837,153.002
C00964=1087.629,44.814,-59.676,174.904,18.838,153.002
C00965=1087.635,45.063,-59.693,174.905,18.840,153.002
C00966=1087.641,45.313,-59.708,174.907,18.842,153.002
C00967=1087.646,45.562,-59.724,174.909,18.843,153.002
C00968=1087.652,45.812,-59.739,174.911,18.846,153.002
C00969=1087.657,46.061,-59.756,174.912,18.848,153.002
C00970=1087.662,46.310,-59.771,174.914,18.849,153.002
C00971=1087.668,46.560,-59.787,174.916,18.851,153.002
C00972=1087.674,46.810,-59.803,174.917,18.853,153.002
C00973=1087.681,47.087,-59.821,174.920,18.855,153.002
C00974=1087.686,47.364,-59.838,174.922,18.857,153.003
C00975=1087.693,47.642,-59.855,174.923,18.859,153.003
C00976=1087.699,47.920,-59.873,174.925,18.861,153.003
C00977=1087.705,48.169,-59.889,174.927,18.862,153.003
C00978=1087.711,48.419,-59.905,174.929,18.865,153.003
C00979=1087.716,48.669,-59.921,174.931,18.866,153.003
C00980=1087.722,48.917,-59.937,174.933,18.869,153.003
C00981=1087.727,49.167,-59.952,174.934,18.870,153.003
C00982=1087.733,49.417,-59.969,174.936,18.872,153.003
C00983=1087.739,49.666,-59.985,174.938,18.874,153.003
C00984=1087.744,49.915,-60.000,174.939,18.875,153.003
C00985=1087.750,50.165,-60.016,174.941,18.877,153.003
C00986=1087.756,50.414,-60.033,174.943,18.879,153.003
C00987=1087.762,50.664,-60.048,174.945,18.881,153.003
C00988=1087.767,50.913,-60.064,174.947,18.882,153.003
C00989=1087.773,51.162,-60.080,174.949,18.884,153.003
C00990=1087.779,51.412,-60.096,174.950,18.886,153.003
C00991=1087.784,51.662,-60.113,174.952,18.888,153.003
C00992=1087.790,51.911,-60.129,174.954,18.890,153.003
C00993=1087.795,52.160,-60.144,174.955,18.892,153.003
C00994=1087.801,52.410,-60.160,174.957,18.894,153.003
C00995=1087.807,52.659,-60.177,174.959,18.895,153.003
C00996=1087.813,52.908,-60.193,174.961,18.897,153.003
C00997=1087.819,53.158,-60.208,174.963,18.899,153.004
C00998=1087.825,53.408,-60.225,174.965,18.901,153.004
C00999=1087.830,53.656,-60.241,174.966,18.902,153.004
C01000=1087.836,53.906,-60.257,174.968,18.904,153.004
C01001=1087.842,54.156,-60.272,174.970,18.906,153.004
C01002=1087.847,54.405,-60.289,174.971,18.908,153.004
C01003=1087.853,54.655,-60.305,174.974,18.910,153.004
C01004=1087.859,54.904,-60.322,174.975,18.911,153.004
C01005=1087.865,55.153,-60.338,174.977,18.913,153.004
C01006=1087.870,55.402,-60.353,174.979,18.915,153.004
C01007=1087.876,55.652,-60.369,174.980,18.916,153.004
C01008=1087.882,55.901,-60.386,174.983,18.918,153.004
C01009=1087.887,56.151,-60.402,174.984,18.920,153.004
C01010=1087.893,56.400,-60.419,174.986,18.922,153.004
C01011=1087.899,56.650,-60.435,174.988,18.923,153.004
C01012=1087.905,56.899,-60.451,174.990,18.925,153.004
C01013=1087.910,57.149,-60.467,174.991,18.927,153.004
C01014=1087.916,57.398,-60.483,174.994,18.929,153.004
C01015=1087.922,57.648,-60.499,174.995,18.931,153.004
C01016=1087.927,57.897,-60.516,174.997,18.933,153.004
C01017=1087.933,58.146,-60.532,174.999,18.934,153.004
C01018=1087.939,58.395,-60.548,175.001,18.935,153.004
C01019=1087.945,58.645,-60.565,175.003,18.937,153.004
C01020=1087.951,58.894,-60.581,175.004,18.939,153.004
C01021=1087.956,59.143,-60.597,175.007,18.941,153.004
C01022=1087.962,59.393,-60.614,175.008,18.942,153.004
C01023=1087.968,59.642,-60.630,175.010,18.944,153.004
C01024=1087.974,59.892,-60.646,175.012,18.946,153.004
C01025=1087.980,60.141,-60.663,175.014,18.948,153.004
C01026=1087.986,60.390,-60.679,175.015,18.949,153.004
C01027=1087.991,60.640,-60.696,175.018,18.952,153.004
C01028=1087.997,60.889,-60.712,175.019,18.953,153.004
C01029=1088.003,61.139,-60.728,175.021,18.954,153.004
C01030=1088.009,61.388,-60.745,175.023,18.956,153.004
C01031=1088.015,61.637,-60.761,175.024,18.958,153.004
C01032=1088.020,61.887,-60.778,175.027,18.960,153.004
C01033=1088.026,62.136,-60.794,175.028,18.961,153.004
C01034=1088.032,62.386,-60.810,175.030,18.963,153.004
C01035=1088.038,62.635,-60.826,175.032,18.965,153.004
C01036=1088.044,62.884,-60.843,175.034,18.966,153.004
C01037=1088.050,63.162,-60.861,175.036,18.968,153.004
C01038=1088.056,63.439,-60.880,175.038,18.970,153.004
C01039=1088.062,63.717,-60.898,175.040,18.972,153.004
C01040=1088.069,63.994,-60.916,175.043,18.974,153.004
C01041=1088.075,64.244,-60.933,175.044,18.976,153.004
C01042=1088.081,64.494,-60.949,175.046,18.978,153.004
C01043=1088.087,64.743,-60.966,175.048,18.979,153.004
C01044=1088.092,64.992,-60.983,175.050,18.981,153.004
C01045=1088.098,65.242,-60.999,175.052,18.982,153.004
C01046=1088.104,65.491,-61.016,175.053,18.984,153.004
C01047=1088.110,65.741,-61.033,175.055,18.986,153.004
C01048=1088.115,65.990,-61.049,175.057,18.987,153.004
C01049=1088.121,66.240,-61.066,175.059,18.989,153.004
C01050=1088.127,66.488,-61.083,175.061,18.991,153.004
C01051=1088.132,66.738,-61.100,175.063,18.993,153.004
C01052=1088.138,66.987,-61.116,175.064,18.995,153.005
C01053=1088.143,67.237,-61.133,175.067,18.996,153.004
C01054=1088.149,67.486,-61.149,175.068,18.998,153.004
C01055=1088.155,67.735,-61.166,175.071,19.000,153.004
C01056=1088.161,67.985,-61.183,175.072,19.001,153.005
C01057=1088.166,68.234,-61.200,175.074,19.003,153.005
C01058=1088.172,68.484,-61.216,175.076,19.005,153.005
C01059=1088.177,68.733,-61.233,175.078,19.007,153.005
C01060=1088.183,68.982,-61.250,175.080,19.008,153.004
C01061=1088.189,69.232,-61.266,175.082,19.010,153.004
C01062=1088.195,69.480,-61.283,175.083,19.011,153.005
C01063=1088.200,69.730,-61.300,175.086,19.013,153.005
C01064=1088.206,69.979,-61.317,175.087,19.015,153.005
C01065=1088.211,70.229,-61.333,175.089,19.017,153.005
C01066=1088.217,70.478,-61.350,175.091,19.018,153.005
C01067=1088.223,70.727,-61.367,175.093,19.020,153.005
C01068=1088.229,70.978,-61.384,175.095,19.022,153.005
C01069=1088.235,71.227,-61.401,175.097,19.024,153.005
C01070=1088.240,71.476,-61.418,175.099,19.025,153.005
C01071=1088.246,71.725,-61.435,175.101,19.027,153.005
C01072=1088.251,71.975,-61.452,175.102,19.028,153.005
C01073=1088.257,72.224,-61.468,175.105,19.030,153.005
C01074=1088.263,72.473,-61.486,175.106,19.032,153.005
C01075=1088.268,72.723,-61.503,175.108,19.034,153.005
C01076=1088.274,72.971,-61.520,175.110,19.035,153.005
C01077=1088.280,73.221,-61.537,175.112,19.037,153.005
C01078=1088.285,73.471,-61.553,175.114,19.038,153.005
C01079=1088.291,73.719,-61.570,175.116,19.041,153.005
C01080=1088.297,73.970,-61.588,175.118,19.042,153.005
C01081=1088.302,74.219,-61.605,175.120,19.044,153.004
C01082=1088.308,74.468,-61.621,175.122,19.045,153.005
C01083=1088.314,74.717,-61.639,175.124,19.047,153.005
C01084=1088.319,74.967,-61.656,175.125,19.049,153.005
C01085=1088.325,75.216,-61.673,175.128,19.051,153.005
C01086=1088.331,75.465,-61.690,175.129,19.052,153.005
C01087=1088.337,75.715,-61.708,175.132,19.054,153.005
C01088=1088.343,75.964,-61.724,175.133,19.055,153.005
C01089=1088.348,76.213,-61.741,175.135,19.057,153.004
C01090=1088.353,76.463,-61.758,175.137,19.058,153.005
C01091=1088.360,76.712,-61.775,175.139,19.060,153.005
C01092=1088.365,76.961,-61.792,175.141,19.062,153.005
C01093=1088.371,77.211,-61.810,175.143,19.064,153.004
C01094=1088.377,77.461,-61.826,175.145,19.065,153.004
C01095=1088.382,77.710,-61.844,175.147,19.067,153.004
C01096=1088.388,77.959,-61.861,175.149,19.068,153.004
C01097=1088.393,78.208,-61.878,175.151,19.070,153.004
C01098=1088.399,78.457,-61.895,175.152,19.072,153.004
C01099=1088.405,78.707,-61.913,175.155,19.074,153.004
C01100=1088.411,78.956,-61.930,175.156,19.075,153.004
C01101=1088.417,79.233,-61.949,175.159,19.077,153.004
C01102=1088.423,79.511,-61.968,175.161,19.079,153.004
C01103=1088.430,79.789,-61.988,175.163,19.081,153.004
C01104=1088.435,80.066,-62.007,175.165,19.083,153.004
C01105=1088.441,80.316,-62.024,175.167,19.084,153.004
C01106=1088.447,80.564,-62.041,175.169,19.086,153.004
C01107=1088.452,80.814,-62.058,175.171,19.088,153.004
C01108=1088.458,81.064,-62.076,175.173,19.089,153.004
C01109=1088.464,81.313,-62.094,175.175,19.091,153.004
C01110=1088.469,81.562,-62.111,175.177,19.093,153.004
C01111=1088.475,81.811,-62.128,175.178,19.094,153.004
C01112=1088.480,82.060,-62.146,175.181,19.096,153.004
C01113=1088.486,82.310,-62.164,175.183,19.098,153.004
C01114=1088.492,82.560,-62.181,175.185,19.099,153.004
C01115=1088.497,82.809,-62.198,175.187,19.101,153.004
C01116=1088.503,83.058,-62.216,175.189,19.102,153.004
C01117=1088.508,83.307,-62.233,175.191,19.104,153.004
C01118=1088.515,83.557,-62.250,175.193,19.105,153.004
C01119=1088.520,83.806,-62.267,175.195,19.107,153.004
C01120=1088.526,84.055,-62.285,175.196,19.109,153.004
C01121=1088.531,84.304,-62.303,175.199,19.111,153.004
C01122=1088.537,84.554,-62.321,175.200,19.112,153.004
C01123=1088.543,84.804,-62.337,175.203,19.114,153.004
C01124=1088.548,85.053,-62.355,175.204,19.115,153.004
C01125=1088.554,85.302,-62.373,175.207,19.117,153.004
C01126=1088.560,85.551,-62.390,175.209,19.119,153.004
C01127=1088.565,85.800,-62.408,175.211,19.120,153.004
C01128=1088.571,86.049,-62.426,175.213,19.122,153.004
C01129=1088.577,86.299,-62.444,175.214,19.123,153.004
C01130=1088.582,86.549,-62.460,175.217,19.125,153.004
C01131=1088.588,86.798,-62.478,175.218,19.126,153.004
C01132=1088.594,87.048,-62.496,175.221,19.128,153.004
C01133=1088.599,87.297,-62.513,175.222,19.129,153.004
C01134=1088.605,87.546,-62.531,175.225,19.131,153.004
C01135=1088.611,87.795,-62.549,175.227,19.133,153.004
C01136=1088.616,88.044,-62.566,175.229,19.135,153.004
C01137=1088.622,88.294,-62.584,175.231,19.137,153.004
C01138=1088.628,88.543,-62.602,175.233,19.138,153.004
C01139=1088.634,88.792,-62.620,175.235,19.140,153.004
C01140=1088.639,89.041,-62.637,175.237,19.141,153.003
C01141=1088.645,89.291,-62.655,175.239,19.143,153.003
C01142=1088.651,89.540,-62.673,175.241,19.144,153.003
C01143=1088.656,89.789,-62.690,175.243,19.146,153.003
C01144=1088.662,90.039,-62.708,175.245,19.147,153.003
C01145=1088.668,90.288,-62.726,175.247,19.149,153.003
C01146=1088.674,90.538,-62.744,175.249,19.150,153.003
C01147=1088.679,90.787,-62.761,175.251,19.152,153.003
C01148=1088.685,91.036,-62.779,175.253,19.153,153.003
C01149=1088.691,91.286,-62.797,175.255,19.155,153.003
C01150=1088.696,91.535,-62.815,175.257,19.157,153.003
C01151=1088.701,91.784,-62.832,175.260,19.159,153.003
C01152=1088.708,92.034,-62.850,175.261,19.160,153.003
C01153=1088.713,92.283,-62.868,175.264,19.162,153.003
C01154=1088.719,92.532,-62.885,175.265,19.163,153.003
C01155=1088.724,92.782,-62.904,175.268,19.165,153.003
C01156=1088.730,93.030,-62.922,175.269,19.166,153.003
C01157=1088.735,93.279,-62.940,175.271,19.168,153.003
C01158=1088.741,93.529,-62.958,175.274,19.169,153.003
C01159=1088.746,93.778,-62.976,175.275,19.171,153.003
C01160=1088.752,94.028,-62.994,175.278,19.172,153.003
C01161=1088.758,94.277,-63.011,175.279,19.174,153.003
C01162=1088.763,94.526,-63.029,175.282,19.175,153.002
C01163=1088.770,94.775,-63.048,175.283,19.177,153.003
C01164=1088.775,95.025,-63.066,175.286,19.178,153.002
C01165=1088.781,95.303,-63.086,175.288,19.181,153.002
C01166=1088.787,95.580,-63.106,175.291,19.182,153.002
C01167=1088.794,95.857,-63.125,175.293,19.184,153.002
C01168=1088.800,96.135,-63.145,175.296,19.186,153.002
C01169=1088.805,96.384,-63.164,175.297,19.187,153.002
C01170=1088.811,96.633,-63.182,175.300,19.189,153.002
C01171=1088.817,96.883,-63.200,175.301,19.190,153.002
C01172=1088.823,97.132,-63.217,175.303,19.192,153.002
C01173=1088.828,97.381,-63.237,175.305,19.193,153.002
C01174=1088.834,97.630,-63.254,175.307,19.195,153.002
C01175=1088.840,97.880,-63.272,175.310,19.196,153.002
C01176=1088.845,98.129,-63.291,175.311,19.198,153.002
C01177=1088.851,98.378,-63.309,175.314,19.199,153.002
C01178=1088.857,98.627,-63.326,175.316,19.200,153.002
C01179=1088.862,98.877,-63.345,175.318,19.202,153.002
C01180=1088.868,99.126,-63.363,175.320,19.204,153.002
C01181=1088.874,99.376,-63.381,175.322,19.206,153.002
C01182=1088.879,99.625,-63.399,175.324,19.207,153.001
C01183=1088.885,99.874,-63.418,175.326,19.208,153.001
C01184=1088.891,100.123,-63.436,175.328,19.210,153.001
C01185=1088.897,100.372,-63.454,175.331,19.212,153.001
C01186=1088.902,100.622,-63.472,175.333,19.213,153.001
C01187=1088.908,100.871,-63.490,175.335,19.215,153.001
C01188=1088.914,101.120,-63.509,175.337,19.216,153.001
C01189=1088.919,101.370,-63.527,175.339,19.217,153.001
C01190=1088.925,101.618,-63.545,175.341,19.219,153.001
C01191=1088.930,101.868,-63.564,175.343,19.220,153.001
C01192=1088.936,102.117,-63.582,175.346,19.222,153.001
C01193=1088.942,102.367,-63.601,175.347,19.223,153.001
C01194=1088.947,102.616,-63.618,175.350,19.225,153.001
C01195=1088.953,102.865,-63.638,175.352,19.226,153.001
C01196=1088.958,103.114,-63.655,175.354,19.228,153.001
C01197=1088.964,103.364,-63.674,175.356,19.230,153.000
C01198=1088.969,103.613,-63.692,175.358,19.232,153.000
C01199=1088.975,103.862,-63.711,175.360,19.233,153.000
C01200=1088.981,104.111,-63.729,175.363,19.234,153.000
C01201=1088.986,104.361,-63.748,175.364,19.236,153.000
C01202=1088.991,104.610,-63.766,175.367,19.237,153.000
C01203=1088.998,104.859,-63.785,175.369,19.239,153.000
C01204=1089.002,105.108,-63.803,175.371,19.240,153.000
C01205=1089.009,105.358,-63.822,175.373,19.242,153.000
C01206=1089.014,105.607,-63.840,175.375,19.243,153.000
C01207=1089.020,105.856,-63.858,175.377,19.244,153.000
C01208=1089.026,106.106,-63.878,175.380,19.246,153.000
C01209=1089.031,106.355,-63.895,175.381,19.247,153.000
C01210=1089.037,106.604,-63.915,175.384,19.249,153.000
C01211=1089.042,106.853,-63.933,175.386,19.251,152.999
C01212=1089.048,107.102,-63.951,175.388,19.252,152.999
C01213=1089.053,107.351,-63.970,175.390,19.254,152.999
C01214=1089.059,107.601,-63.988,175.393,19.255,152.999
C01215=1089.065,107.850,-64.007,175.395,19.256,152.999
C01216=1089.071,108.099,-64.026,175.397,19.258,152.999
C01217=1089.076,108.349,-64.044,175.398,19.259,152.999
C01218=1089.081,108.598,-64.063,175.401,19.261,152.999
C01219=1089.088,108.847,-64.082,175.404,19.262,152.999
C01220=1089.093,109.097,-64.100,175.405,19.263,152.999
C01221=1089.099,109.345,-64.119,175.408,19.265,152.999
C01222=1089.105,109.595,-64.138,175.410,19.267,152.999
C01223=1089.110,109.845,-64.156,175.412,19.268,152.998
C01224=1089.116,110.093,-64.175,175.414,19.269,152.998
C01225=1089.122,110.343,-64.194,175.416,19.270,152.998
C01226=1089.127,110.592,-64.213,175.418,19.272,152.998
C01227=1089.133,110.841,-64.231,175.421,19.274,152.998
C01228=1089.138,111.090,-64.250,175.422,19.275,152.998
C01229=1089.145,111.368,-64.271,175.425,19.277,152.998
C01230=1089.151,111.645,-64.292,175.428,19.278,152.998
C01231=1089.158,111.923,-64.313,175.430,19.280,152.998
C01232=1089.163,112.201,-64.334,175.433,19.281,152.998
C01233=1089.169,112.449,-64.352,175.435,19.283,152.998
C01234=1089.175,112.699,-64.371,175.437,19.285,152.997
C01235=1089.181,112.948,-64.391,175.439,19.286,152.997
C01236=1089.186,113.196,-64.409,175.442,19.287,152.997
C01237=1089.192,113.446,-64.427,175.443,19.288,152.997
C01238=1089.197,113.696,-64.447,175.446,19.290,152.997
C01239=1089.203,113.945,-64.466,175.448,19.291,152.997
C01240=1089.208,114.194,-64.485,175.450,19.293,152.997
C01241=1089.215,114.443,-64.503,175.452,19.294,152.997
C01242=1089.220,114.693,-64.523,175.455,19.296,152.997
C01243=1089.225,114.941,-64.541,175.457,19.297,152.997
C01244=1089.231,115.191,-64.561,175.459,19.299,152.996
C01245=1089.237,115.440,-64.580,175.462,19.300,152.996
C01246=1089.242,115.689,-64.599,175.463,19.302,152.996
C01247=1089.247,115.939,-64.617,175.466,19.303,152.996
C01248=1089.253,116.188,-64.637,175.468,19.305,152.996
C01249=1089.258,116.437,-64.655,175.470,19.306,152.996
C01250=1089.264,116.687,-64.675,175.472,19.307,152.996
C01251=1089.269,116.936,-64.694,175.475,19.309,152.996
C01252=1089.275,117.185,-64.713,175.476,19.310,152.996
C01253=1089.280,117.434,-64.732,175.479,19.312,152.996
C01254=1089.287,117.683,-64.751,175.481,19.313,152.996
C01255=1089.292,117.932,-64.770,175.483,19.314,152.995
C01256=1089.297,118.181,-64.789,175.486,19.316,152.995
C01257=1089.303,118.431,-64.808,175.488,19.318,152.995
C01258=1089.308,118.680,-64.827,175.491,19.319,152.995
C01259=1089.314,118.929,-64.846,175.492,19.320,152.995
C01260=1089.320,119.178,-64.866,175.495,19.322,152.995
C01261=1089.326,119.427,-64.885,175.497,19.324,152.995
C01262=1089.331,119.676,-64.904,175.499,19.325,152.995
C01263=1089.336,119.925,-64.924,175.501,19.326,152.995
C01264=1089.342,120.175,-64.943,175.504,19.328,152.995
C01265=1089.348,120.424,-64.962,175.506,19.329,152.994
C01266=1089.353,120.673,-64.981,175.508,19.330,152.994
C01267=1089.359,120.923,-65.000,175.511,19.332,152.994
C01268=1089.364,121.172,-65.019,175.512,19.333,152.994
C01269=1089.370,121.421,-65.039,175.515,19.334,152.994
C01270=1089.376,121.670,-65.059,175.517,19.336,152.994
C01271=1089.381,121.919,-65.077,175.519,19.337,152.994
C01272=1089.387,122.168,-65.097,175.522,19.339,152.994
C01273=1089.392,122.418,-65.116,175.524,19.340,152.994
C01274=1089.397,122.668,-65.136,175.526,19.341,152.993
C01275=1089.403,122.916,-65.156,175.528,19.343,152.993
C01276=1089.408,123.165,-65.175,175.531,19.344,152.993
C01277=1089.414,123.415,-65.194,175.533,19.346,152.993
C01278=1089.420,123.664,-65.213,175.535,19.347,152.993
C01279=1089.426,123.913,-65.233,175.538,19.348,152.993
C01280=1089.431,124.162,-65.252,175.540,19.350,152.993
C01281=1089.437,124.412,-65.272,175.542,19.351,152.993
C01282=1089.442,124.660,-65.290,175.544,19.352,152.993
C01283=1089.448,124.909,-65.310,175.547,19.353,152.992
C01284=1089.454,125.159,-65.330,175.549,19.354,152.992
C01285=1089.460,125.408,-65.349,175.551,19.356,152.992
C01286=1089.466,125.657,-65.369,175.554,19.357,152.992
C01287=1089.471,125.906,-65.388,175.556,19.359,152.992
C01288=1089.476,126.156,-65.408,175.558,19.360,152.992
C01289=1089.482,126.405,-65.428,175.561,19.362,152.992
C01290=1089.487,126.654,-65.447,175.563,19.363,152.991
C01291=1089.493,126.903,-65.466,175.565,19.364,152.991
C01292=1089.499,127.152,-65.486,175.568,19.365,152.991
C01293=1089.506,127.430,-65.508,175.570,19.367,152.991
C01294=1089.511,127.708,-65.529,175.573,19.368,152.991
C01295=1089.518,127.985,-65.551,175.575,19.370,152.991
C01296=1089.524,128.262,-65.573,175.578,19.371,152.991
C01297=1089.530,128.511,-65.593,175.580,19.373,152.990
C01298=1089.535,128.760,-65.612,175.583,19.374,152.990
C01299=1089.541,129.009,-65.632,175.585,19.375,152.990
C01300=1089.547,129.259,-65.651,175.587,19.376,152.990
C01301=1089.553,129.508,-65.671,175.590,19.378,152.990
C01302=1089.559,129.757,-65.690,175.592,19.380,152.990
C01303=1089.564,130.007,-65.710,175.594,19.380,152.990
C01304=1089.570,130.256,-65.730,175.597,19.382,152.989
C01305=1089.575,130.505,-65.749,175.599,19.383,152.989
C01306=1089.581,130.754,-65.769,175.601,19.384,152.989
C01307=1089.587,131.003,-65.789,175.604,19.385,152.989
C01308=1089.593,131.252,-65.809,175.606,19.387,152.989
C01309=1089.598,131.501,-65.829,175.609,19.388,152.989
C01310=1089.604,131.751,-65.848,175.611,19.389,152.989
C01311=1089.610,131.999,-65.868,175.613,19.390,152.988
C01312=1089.616,132.249,-65.888,175.616,19.392,152.988
C01313=1089.621,132.498,-65.908,175.618,19.393,152.988
C01314=1089.627,132.747,-65.927,175.620,19.394,152.988
C01315=1089.633,132.996,-65.947,175.623,19.396,152.988
C01316=1089.638,133.245,-65.968,175.625,19.397,152.988
C01317=1089.644,133.495,-65.987,175.628,19.399,152.987
C01318=1089.650,133.744,-66.007,175.630,19.400,152.987
C01319=1089.654,133.993,-66.027,175.632,19.401,152.987
C01320=1089.660,134.242,-66.047,175.635,19.402,152.987
C01321=1089.666,134.491,-66.068,175.637,19.403,152.987
C01322=1089.671,134.741,-66.087,175.639,19.405,152.987
C01323=1089.677,134.989,-66.107,175.642,19.406,152.987
C01324=1089.683,135.239,-66.127,175.644,19.408,152.987
C01325=1089.688,135.488,-66.147,175.646,19.408,152.986
C01326=1089.694,135.737,-66.167,175.649,19.410,152.986
C01327=1089.700,135.986,-66.187,175.651,19.411,152.986
C01328=1089.706,136.235,-66.207,175.654,19.412,152.986
C01329=1089.711,136.485,-66.227,175.657,19.414,152.986
C01330=1089.717,136.733,-66.247,175.658,19.415,152.986
C01331=1089.722,136.982,-66.267,175.661,19.417,152.985
C01332=1089.728,137.231,-66.287,175.664,19.418,152.985
C01333=1089.733,137.481,-66.307,175.666,19.419,152.985
C01334=1089.739,137.730,-66.327,175.668,19.420,152.985
C01335=1089.744,137.979,-66.348,175.671,19.421,152.985
C01336=1089.750,138.228,-66.368,175.673,19.423,152.985
C01337=1089.756,138.477,-66.388,175.676,19.424,152.984
C01338=1089.761,138.726,-66.407,175.678,19.425,152.984
C01339=1089.767,138.975,-66.427,175.680,19.426,152.984
C01340=1089.772,139.224,-66.448,175.683,19.428,152.984
C01341=1089.777,139.473,-66.468,175.685,19.429,152.984
C01342=1089.784,139.723,-66.489,175.687,19.430,152.984
C01343=1089.789,139.972,-66.509,175.690,19.431,152.984
C01344=1089.795,140.221,-66.529,175.692,19.433,152.983
C01345=1089.800,140.471,-66.549,175.695,19.434,152.983
C01346=1089.806,140.719,-66.569,175.697,19.436,152.983
C01347=1089.811,140.969,-66.590,175.699,19.436,152.983
C01348=1089.817,141.217,-66.610,175.702,19.438,152.983
C01349=1089.823,141.466,-66.630,175.704,19.439,152.983
C01350=1089.828,141.716,-66.651,175.707,19.440,152.982
C01351=1089.834,141.964,-66.671,175.709,19.441,152.982
C01352=1089.839,142.214,-66.691,175.711,19.443,152.982
C01353=1089.845,142.463,-66.712,175.714,19.444,152.982
C01354=1089.851,142.712,-66.732,175.717,19.445,152.982
C01355=1089.856,142.961,-66.753,175.720,19.446,152.981
C01356=1089.862,143.210,-66.773,175.721,19.447,152.981
C01357=1089.868,143.487,-66.795,175.724,19.449,152.981
C01358=1089.874,143.765,-66.819,175.727,19.451,152.981
C01359=1089.880,144.042,-66.841,175.730,19.452,152.981
C01360=1089.886,144.320,-66.864,175.733,19.453,152.980
C01361=1089.892,144.569,-66.884,175.735,19.455,152.980
C01362=1089.898,144.818,-66.904,175.737,19.455,152.980
C01363=1089.903,145.067,-66.925,175.740,19.457,152.980
C01364=1089.909,145.316,-66.945,175.742,19.458,152.980
C01365=1089.915,145.565,-66.966,175.745,19.459,152.980
C01366=1089.920,145.814,-66.987,175.747,19.461,152.980
C01367=1089.926,146.063,-67.007,175.749,19.461,152.979
C01368=1089.932,146.312,-67.028,175.752,19.463,152.979
C01369=1089.937,146.562,-67.048,175.755,19.464,152.979
C01370=1089.943,146.811,-67.068,175.757,19.466,152.979
C01371=1089.949,147.060,-67.089,175.760,19.467,152.979
C01372=1089.954,147.309,-67.110,175.762,19.468,152.978
C01373=1089.959,147.558,-67.131,175.764,19.469,152.978
C01374=1089.965,147.807,-67.151,175.767,19.470,152.978
C01375=1089.971,148.056,-67.172,175.770,19.471,152.978
C01376=1089.977,148.306,-67.192,175.772,19.473,152.978
C01377=1089.982,148.555,-67.213,175.774,19.473,152.977
C01378=1089.987,148.803,-67.234,175.777,19.475,152.977
C01379=1089.994,149.053,-67.254,175.780,19.476,152.977
C01380=1089.999,149.302,-67.275,175.782,19.477,152.977
C01381=1090.004,149.551,-67.295,175.785,19.478,152.977
C01382=1090.010,149.799,-67.317,175.787,19.480,152.977
C01383=1090.015,150.049,-67.337,175.789,19.481,152.976
C01384=1090.021,150.298,-67.358,175.792,19.482,152.976
C01385=1090.026,150.548,-67.379,175.795,19.483,152.976
C01386=1090.033,150.796,-67.399,175.797,19.485,152.976
C01387=1090.038,151.045,-67.420,175.800,19.486,152.976
C01388=1090.044,151.295,-67.441,175.802,19.487,152.975
C01389=1090.049,151.543,-67.462,175.804,19.488,152.975
C01390=1090.055,151.792,-67.483,175.807,19.489,152.975
C01391=1090.060,152.041,-67.503,175.810,19.490,152.975
C01392=1090.066,152.291,-67.525,175.812,19.491,152.975
C01393=1090.071,152.540,-67.545,175.815,19.493,152.974
C01394=1090.077,152.789,-67.566,175.818,19.494,152.974
C01395=1090.082,153.037,-67.587,175.819,19.495,152.974
C01396=1090.088,153.287,-67.608,175.822,19.496,152.974
C01397=1090.094,153.536,-67.629,175.825,19.498,152.974
C01398=1090.099,153.785,-67.650,175.828,19.499,152.973
C01399=1090.105,154.034,-67.670,175.830,19.500,152.973
C01400=1090.111,154.283,-67.692,175.833,19.501,152.973
C01401=1090.116,154.532,-67.712,175.835,19.502,152.973
C01402=1090.122,154.781,-67.734,175.837,19.503,152.973
C01403=1090.128,155.030,-67.754,175.840,19.504,152.972
C01404=1090.133,155.279,-67.776,175.843,19.505,152.972
C01405=1090.139,155.529,-67.797,175.845,19.507,152.972
C01406=1090.145,155.777,-67.818,175.848,19.508,152.972
C01407=1090.150,156.026,-67.838,175.851,19.509,152.972
C01408=1090.156,156.275,-67.860,175.853,19.510,152.971
C01409=1090.161,156.525,-67.881,175.855,19.511,152.971
C01410=1090.166,156.773,-67.902,175.858,19.513,152.971
C01411=1090.172,157.023,-67.923,175.861,19.514,152.971
C01412=1090.178,157.272,-67.945,175.863,19.515,152.971
C01413=1090.183,157.520,-67.966,175.866,19.516,152.970
C01414=1090.189,157.770,-67.987,175.869,19.517,152.970
C01415=1090.195,158.019,-68.008,175.871,19.518,152.970
C01416=1090.200,158.268,-68.029,175.873,19.519,152.970
C01417=1090.206,158.517,-68.050,175.876,19.520,152.970
C01418=1090.212,158.765,-68.072,175.879,19.522,152.969
C01419=1090.217,159.015,-68.092,175.881,19.523,152.969
C01420=1090.222,159.264,-68.114,175.884,19.524,152.969
C01421=1090.229,159.541,-68.138,175.887,19.525,152.969
C01422=1090.235,159.818,-68.161,175.889,19.527,152.969
C01423=1090.242,160.095,-68.185,175.892,19.528,152.968
C01424=1090.248,160.372,-68.209,175.896,19.529,152.968
C01425=1090.253,160.622,-68.230,175.898,19.530,152.968
C01426=1090.258,160.870,-68.251,175.900,19.531,152.968
C01427=1090.264,161.120,-68.273,175.903,19.532,152.967
C01428=1090.270,161.369,-68.293,175.906,19.533,152.967
C01429=1090.276,161.618,-68.315,175.909,19.535,152.967
C01430=1090.281,161.867,-68.337,175.911,19.536,152.967
C01431=1090.286,162.115,-68.358,175.914,19.537,152.966
C01432=1090.292,162.365,-68.379,175.917,19.538,152.966
C01433=1090.297,162.614,-68.401,175.918,19.539,152.966
C01434=1090.302,162.862,-68.422,175.921,19.540,152.966
C01435=1090.308,163.112,-68.444,175.924,19.542,152.966
C01436=1090.313,163.360,-68.466,175.926,19.543,152.966
C01437=1090.319,163.610,-68.487,175.929,19.544,152.965
C01438=1090.324,163.859,-68.508,175.932,19.545,152.965
C01439=1090.330,164.108,-68.530,175.934,19.546,152.965
C01440=1090.335,164.357,-68.552,175.937,19.548,152.965
C01441=1090.341,164.606,-68.573,175.940,19.549,152.964
C01442=1090.347,164.855,-68.595,175.943,19.550,152.964
C01443=1090.352,165.104,-68.617,175.945,19.551,152.964
C01444=1090.357,165.353,-68.637,175.947,19.552,152.964
C01445=1090.362,165.602,-68.659,175.950,19.553,152.964
C01446=1090.368,165.851,-68.681,175.953,19.554,152.963
C01447=1090.373,166.100,-68.703,175.955,19.556,152.963
C01448=1090.379,166.349,-68.724,175.958,19.557,152.963
C01449=1090.385,166.598,-68.746,175.961,19.558,152.963
C01450=1090.390,166.847,-68.768,175.963,19.559,152.962
C01451=1090.396,167.096,-68.789,175.966,19.561,152.962
C01452=1090.401,167.345,-68.811,175.969,19.562,152.962
C01453=1090.406,167.593,-68.833,175.972,19.563,152.962
C01454=1090.412,167.843,-68.855,175.974,19.564,152.962
C01455=1090.417,168.091,-68.876,175.977,19.565,152.961
C01456=1090.423,168.341,-68.898,175.979,19.566,152.961
C01457=1090.428,168.589,-68.920,175.982,19.567,152.961
C01458=1090.434,168.839,-68.942,175.984,19.568,152.961
C01459=1090.439,169.087,-68.963,175.987,19.569,152.961
C01460=1090.445,169.337,-68.985,175.990,19.570,152.960
C01461=1090.450,169.585,-69.007,175.992,19.572,152.960
C01462=1090.456,169.835,-69.029,175.995,19.573,152.960
C01463=1090.462,170.084,-69.050,175.998,19.574,152.960
C01464=1090.467,170.333,-69.072,176.000,19.575,152.959
C01465=1090.473,170.582,-69.094,176.003,19.576,152.959
C01466=1090.478,170.830,-69.116,176.006,19.577,152.959
C01467=1090.484,171.080,-69.138,176.009,19.578,152.959
C01468=1090.489,171.328,-69.160,176.012,19.579,152.958
C01469=1090.495,171.578,-69.182,176.014,19.580,152.958
C01470=1090.500,171.826,-69.203,176.016,19.581,152.958
C01471=1090.505,172.076,-69.226,176.019,19.583,152.958
C01472=1090.512,172.324,-69.248,176.022,19.584,152.958
C01473=1090.517,172.573,-69.270,176.024,19.585,152.957
C01474=1090.523,172.822,-69.292,176.027,19.586,152.957
C01475=1090.528,173.071,-69.313,176.030,19.587,152.957
C01476=1090.534,173.320,-69.335,176.033,19.588,152.957
C01477=1090.540,173.569,-69.358,176.035,19.589,152.956
C01478=1090.544,173.818,-69.380,176.038,19.590,152.956
C01479=1090.551,174.067,-69.401,176.041,19.591,152.956
C01480=1090.556,174.317,-69.424,176.043,19.592,152.956
C01481=1090.562,174.565,-69.446,176.046,19.594,152.955
C01482=1090.567,174.814,-69.468,176.049,19.595,152.955
C01483=1090.572,175.063,-69.490,176.052,19.596,152.955
C01484=1090.579,175.312,-69.512,176.055,19.597,152.955
C01485=1090.584,175.589,-69.537,176.057,19.598,152.954
C01486=1090.591,175.866,-69.561,176.060,19.599,152.954
C01487=1090.597,176.142,-69.585,176.064,19.600,152.954
C01488=1090.603,176.419,-69.610,176.066,19.601,152.954
C01489=1090.609,176.668,-69.632,176.069,19.602,152.953
C01490=1090.615,176.917,-69.655,176.072,19.604,152.953
C01491=1090.620,177.166,-69.677,176.075,19.605,152.953
C01492=1090.626,177.415,-69.699,176.078,19.606,152.953
C01493=1090.632,177.664,-69.722,176.080,19.607,152.952
C01494=1090.637,177.913,-69.743,176.083,19.608,152.952
C01495=1090.643,178.162,-69.766,176.086,19.609,152.952
C01496=1090.648,178.411,-69.788,176.089,19.610,152.952
C01497=1090.654,178.660,-69.811,176.091,19.611,152.951
C01498=1090.660,178.909,-69.832,176.094,19.612,152.951
C01499=1090.665,179.157,-69.855,176.097,19.613,152.951
C01500=1090.671,179.407,-69.877,176.100,19.614,152.950
C01501=1090.677,179.656,-69.900,176.103,19.615,152.950
C01502=1090.682,179.904,-69.922,176.106,19.616,152.950
C01503=1090.688,180.153,-69.945,176.108,19.617,152.950
C01504=1090.694,180.402,-69.966,176.111,19.618,152.949
C01505=1090.700,180.651,-69.989,176.114,19.619,152.949
C01506=1090.705,180.901,-70.011,176.117,19.620,152.949
C01507=1090.710,181.149,-70.034,176.119,19.621,152.949
C01508=1090.717,181.398,-70.056,176.122,19.622,152.948
C01509=1090.722,181.647,-70.078,176.125,19.623,152.948
C01510=1090.728,181.896,-70.101,176.128,19.624,152.948
C01511=1090.734,182.145,-70.123,176.131,19.625,152.947
C01512=1090.739,182.393,-70.146,176.133,19.626,152.947
C01513=1090.745,182.642,-70.169,176.136,19.627,152.947
C01514=1090.750,182.892,-70.191,176.139,19.628,152.947
C01515=1090.757,183.140,-70.213,176.142,19.629,152.946
C01516=1090.763,183.389,-70.236,176.145,19.630,152.946
C01517=1090.768,183.639,-70.258,176.148,19.631,152.946
C01518=1090.773,183.887,-70.281,176.150,19.632,152.945
C01519=1090.780,184.136,-70.303,176.153,19.633,152.945
C01520=1090.785,184.385,-70.326,176.156,19.634,152.945
C01521=1090.791,184.634,-70.348,176.159,19.635,152.945
C01522=1090.797,184.883,-70.371,176.161,19.636,152.944
C01523=1090.803,185.132,-70.394,176.164,19.636,152.944
C01524=1090.808,185.381,-70.417,176.167,19.638,152.944
C01525=1090.813,185.630,-70.439,176.170,19.639,152.944
C01526=1090.819,185.878,-70.462,176.173,19.640,152.943
C01527=1090.824,186.127,-70.485,176.175,19.641,152.943
C01528=1090.830,186.377,-70.507,176.178,19.642,152.943
C01529=1090.835,186.625,-70.530,176.181,19.643,152.943
C01530=1090.841,186.874,-70.553,176.184,19.644,152.942
C01531=1090.846,187.123,-70.576,176.186,19.645,152.942
C01532=1090.852,187.372,-70.599,176.189,19.646,152.942
C01533=1090.858,187.621,-70.622,176.192,19.647,152.941
C01534=1090.862,187.870,-70.644,176.195,19.648,152.941
C01535=1090.868,188.119,-70.667,176.198,19.649,152.941
C01536=1090.873,188.368,-70.690,176.200,19.650,152.941
C01537=1090.879,188.616,-70.713,176.203,19.651,152.940
C01538=1090.885,188.865,-70.736,176.206,19.652,152.940
C01539=1090.890,189.114,-70.759,176.209,19.653,152.940
C01540=1090.896,189.362,-70.781,176.212,19.654,152.940
C01541=1090.901,189.612,-70.805,176.214,19.656,152.939
C01542=1090.906,189.861,-70.828,176.217,19.657,152.939
C01543=1090.912,190.109,-70.851,176.221,19.658,152.939
C01544=1090.918,190.358,-70.874,176.223,19.659,152.939
C01545=1090.924,190.607,-70.897,176.226,19.660,152.938
C01546=1090.929,190.856,-70.920,176.229,19.661,152.938
C01547=1090.934,191.105,-70.943,176.232,19.662,152.938
C01548=1090.939,191.354,-70.966,176.235,19.663,152.938
C01549=1090.945,191.631,-70.991,176.238,19.664,152.937
C01550=1090.952,191.907,-71.017,176.241,19.666,152.937
C01551=1090.958,192.183,-71.043,176.244,19.667,152.937
C01552=1090.964,192.460,-71.069,176.247,19.668,152.936
C01553=1090.970,192.709,-71.091,176.251,19.669,152.936
C01554=1090.976,192.958,-71.114,176.253,19.670,152.936
C01555=1090.981,193.206,-71.137,176.256,19.671,152.936
C01556=1090.986,193.456,-71.161,176.259,19.672,152.935
C01557=1090.992,193.705,-71.184,176.262,19.673,152.935
C01558=1090.997,193.953,-71.206,176.264,19.674,152.935
C01559=1091.003,194.202,-71.229,176.267,19.675,152.934
C01560=1091.008,194.451,-71.253,176.270,19.676,152.934
C01561=1091.014,194.699,-71.277,176.273,19.677,152.934
C01562=1091.020,194.948,-71.300,176.276,19.678,152.934
C01563=1091.026,195.197,-71.322,176.278,19.679,152.933
C01564=1091.031,195.446,-71.346,176.281,19.680,152.933
C01565=1091.036,195.695,-71.369,176.285,19.681,152.933
C01566=1091.042,195.943,-71.393,176.288,19.682,152.932
C01567=1091.048,196.192,-71.416,176.291,19.683,152.932
C01568=1091.053,196.441,-71.439,176.293,19.684,152.932
C01569=1091.059,196.690,-71.462,176.296,19.685,152.932
C01570=1091.065,196.939,-71.486,176.299,19.686,152.931
C01571=1091.071,197.188,-71.509,176.302,19.687,152.931
C01572=1091.076,197.437,-71.533,176.305,19.688,152.931
C01573=1091.082,197.686,-71.556,176.308,19.689,152.931
C01574=1091.088,197.935,-71.579,176.311,19.690,152.930
C01575=1091.093,198.184,-71.603,176.313,19.691,152.930
C01576=1091.099,198.433,-71.626,176.317,19.692,152.930
C01577=1091.105,198.681,-71.649,176.320,19.693,152.929
C01578=1091.110,198.930,-71.673,176.323,19.694,152.929
C01579=1091.115,199.179,-71.696,176.325,19.695,152.929
C01580=1091.121,199.427,-71.719,176.328,19.696,152.928
C01581=1091.126,199.677,-71.743,176.331,19.697,152.928
C01582=1091.132,199.925,-71.767,176.334,19.698,152.928
C01583=1091.138,200.174,-71.790,176.337,19.699,152.928
C01584=1091.144,200.424,-71.814,176.340,19.699,152.927
C01585=1091.150,200.672,-71.837,176.343,19.701,152.927
C01586=1091.156,200.921,-71.860,176.346,19.702,152.927
C01587=1091.161,201.169,-71.884,176.349,19.703,152.926
C01588=1091.167,201.418,-71.907,176.352,19.704,152.926
C01589=1091.172,201.667,-71.932,176.355,19.705,152.926
C01590=1091.178,201.916,-71.955,176.357,19.706,152.926
C01591=1091.184,202.165,-71.979,176.360,19.707,152.925
C01592=1091.189,202.414,-72.002,176.363,19.708,152.925
C01593=1091.195,202.662,-72.026,176.367,19.709,152.924
C01594=1091.200,202.911,-72.049,176.370,19.710,152.924
C01595=1091.206,203.160,-72.073,176.373,19.711,152.924
C01596=1091.211,203.409,-72.097,176.375,19.712,152.924
C01597=1091.217,203.657,-72.120,176.378,19.713,152.923
C01598=1091.223,203.907,-72.145,176.381,19.714,152.923
C01599=1091.228,204.156,-72.168,176.384,19.715,152.923
C01600=1091.234,204.404,-72.192,176.388,19.716,152.923
C01601=1091.239,204.653,-72.216,176.390,19.717,152.922
C01602=1091.245,204.901,-72.239,176.393,19.718,152.922
C01603=1091.251,205.150,-72.263,176.396,19.719,152.922
C01604=1091.256,205.399,-72.287,176.399,19.720,152.921
C01605=1091.262,205.648,-72.311,176.402,19.721,152.921
C01606=1091.268,205.897,-72.335,176.405,19.722,152.921
C01607=1091.273,206.146,-72.358,176.408,19.723,152.920
C01608=1091.279,206.394,-72.382,176.411,19.724,152.920
C01609=1091.284,206.643,-72.407,176.414,19.725,152.920
C01610=1091.290,206.892,-72.430,176.417,19.726,152.920
C01611=1091.295,207.141,-72.454,176.420,19.727,152.919
C01612=1091.301,207.390,-72.479,176.423,19.728,152.919
C01613=1091.324,208.410,-72.576,176.487,19.759,152.915
C01614=1091.332,208.789,-72.613,176.491,19.762,152.914
C01615=1091.341,209.168,-72.651,176.495,19.765,152.914
C01616=1091.350,209.547,-72.687,176.501,19.768,152.914
C01617=1091.358,209.925,-72.725,176.505,19.771,152.914
C01618=1091.364,210.174,-72.750,176.507,19.772,152.914
C01619=1091.370,210.423,-72.773,176.510,19.774,152.914
C01620=1091.376,210.672,-72.798,176.513,19.777,152.914
C01621=1091.381,210.920,-72.822,176.516,19.779,152.914
C01622=1091.386,211.169,-72.846,176.519,19.780,152.914
C01623=1091.392,211.418,-72.871,176.522,19.782,152.914
C01624=1091.397,211.667,-72.895,176.524,19.784,152.914
C01625=1091.403,211.915,-72.920,176.528,19.786,152.914
C01626=1091.409,212.164,-72.945,176.530,19.788,152.913
C01627=1091.414,212.413,-72.969,176.533,19.790,152.913
C01628=1091.420,212.662,-72.994,176.536,19.792,152.913
C01629=1091.425,212.911,-73.018,176.538,19.793,152.913
C01630=1091.431,213.159,-73.043,176.542,19.796,152.913
C01631=1091.437,213.408,-73.068,176.544,19.798,152.913
C01632=1091.442,213.656,-73.092,176.547,19.800,152.913
C01633=1091.448,213.906,-73.117,176.550,19.801,152.913
C01634=1091.454,214.154,-73.142,176.553,19.804,152.913
C01635=1091.459,214.402,-73.166,176.556,19.805,152.913
C01636=1091.465,214.652,-73.190,176.559,19.807,152.913
C01637=1091.470,214.900,-73.216,176.561,19.809,152.913
C01638=1091.476,215.149,-73.241,176.565,19.811,152.913
C01639=1091.481,215.398,-73.265,176.567,19.813,152.912
C01640=1091.487,215.646,-73.290,176.570,19.816,152.913
C01641=1091.492,215.895,-73.314,176.573,19.817,152.912
C01642=1091.498,216.144,-73.339,176.576,19.819,152.912
C01643=1091.504,216.392,-73.364,176.579,19.821,152.912
C01644=1091.509,216.641,-73.389,176.582,19.823,152.912
C01645=1091.514,216.890,-73.413,176.585,19.825,152.912
C01646=1091.520,217.138,-73.438,176.588,19.827,152.912
C01647=1091.526,217.388,-73.463,176.590,19.829,152.912
C01648=1091.532,217.636,-73.488,176.594,19.831,152.912
C01649=1091.537,217.885,-73.513,176.596,19.833,152.912
C01650=1091.542,218.133,-73.538,176.599,19.835,152.912
C01651=1091.548,218.383,-73.563,176.602,19.837,152.912
C01652=1091.554,218.630,-73.588,176.605,19.839,152.912
C01653=1091.560,218.880,-73.612,176.607,19.841,152.912
C01654=1091.566,219.128,-73.638,176.611,19.843,152.911
C01655=1091.570,219.377,-73.663,176.613,19.844,152.911
C01656=1091.577,219.626,-73.688,176.617,19.846,152.911
C01657=1091.582,219.875,-73.712,176.619,19.848,152.911
C01658=1091.588,220.123,-73.738,176.622,19.850,152.911
C01659=1091.594,220.371,-73.763,176.625,19.852,152.911
C01660=1091.599,220.621,-73.788,176.628,19.854,152.911
C01661=1091.605,220.869,-73.813,176.631,19.856,152.911
C01662=1091.610,221.118,-73.837,176.634,19.858,152.911
C01663=1091.617,221.367,-73.863,176.637,19.860,152.911
C01664=1091.622,221.615,-73.888,176.640,19.862,152.911
C01665=1091.627,221.864,-73.913,176.642,19.864,152.911
C01666=1091.636,222.247,-73.951,176.647,19.867,152.910
C01667=1091.645,222.629,-73.991,176.651,19.870,152.910
C01668=1091.653,223.012,-74.030,176.656,19.873,152.910
C01669=1091.662,223.395,-74.068,176.660,19.876,152.910
C01670=1091.667,223.644,-74.094,176.663,19.878,152.910
C01671=1091.673,223.892,-74.119,176.666,19.880,152.910
C01672=1091.679,224.141,-74.144,176.669,19.882,152.910
C01673=1091.684,224.390,-74.169,176.672,19.884,152.910
C01674=1091.690,224.638,-74.194,176.675,19.886,152.910
C01675=1091.695,224.887,-74.220,176.678,19.888,152.910
C01676=1091.701,225.135,-74.245,176.681,19.890,152.910
C01677=1091.707,225.384,-74.271,176.683,19.892,152.910
C01678=1091.712,225.633,-74.296,176.687,19.894,152.910
C01679=1091.717,225.882,-74.321,176.689,19.896,152.910
C01680=1091.723,226.130,-74.347,176.692,19.898,152.910
C01681=1091.729,226.379,-74.373,176.695,19.900,152.909
C01682=1091.735,226.627,-74.398,176.698,19.902,152.909
C01683=1091.740,226.876,-74.424,176.701,19.904,152.909
C01684=1091.746,227.125,-74.449,176.704,19.906,152.909
C01685=1091.751,227.373,-74.474,176.707,19.908,152.909
C01686=1091.757,227.622,-74.500,176.710,19.910,152.909
C01687=1091.763,227.871,-74.526,176.713,19.912,152.909
C01688=1091.768,228.119,-74.551,176.716,19.914,152.909
C01689=1091.774,228.368,-74.577,176.719,19.916,152.909
C01690=1091.780,228.617,-74.602,176.721,19.918,152.909
C01691=1091.786,228.866,-74.628,176.725,19.920,152.909
C01692=1091.791,229.113,-74.653,176.728,19.922,152.909
C01693=1091.797,229.362,-74.679,176.730,19.924,152.909
C01694=1091.803,229.611,-74.704,176.734,19.926,152.909
C01695=1091.808,229.860,-74.730,176.736,19.928,152.909
C01696=1091.813,230.108,-74.756,176.739,19.930,152.909
C01697=1091.819,230.357,-74.781,176.742,19.932,152.908
C01698=1091.825,230.606,-74.807,176.745,19.934,152.908
C01699=1091.831,230.855,-74.832,176.748,19.936,152.908
C01700=1091.836,231.103,-74.858,176.751,19.938,152.908
C01701=1091.841,231.352,-74.884,176.754,19.940,152.908
C01702=1091.847,231.601,-74.910,176.757,19.942,152.908
C01703=1091.853,231.849,-74.936,176.760,19.944,152.908
C01704=1091.858,232.097,-74.961,176.762,19.946,152.908
C01705=1091.864,232.346,-74.987,176.766,19.948,152.908
C01706=1091.870,232.595,-75.013,176.769,19.951,152.908
C01707=1091.875,232.844,-75.038,176.771,19.952,152.908
C01708=1091.881,233.092,-75.065,176.775,19.954,152.908
C01709=1091.886,233.341,-75.091,176.777,19.956,152.908
C01710=1091.892,233.589,-75.116,176.780,19.958,152.908
C01711=1091.898,233.838,-75.142,176.784,19.960,152.908
C01712=1091.903,234.087,-75.169,176.786,19.962,152.908
C01713=1091.909,234.336,-75.195,176.790,19.964,152.907
C01714=1091.914,234.585,-75.220,176.792,19.966,152.908
C01715=1091.920,234.832,-75.246,176.795,19.968,152.907
C01716=1091.926,235.081,-75.272,176.798,19.971,152.907
C01717=1091.931,235.330,-75.298,176.801,19.973,152.907
C01718=1091.940,235.704,-75.337,176.806,19.976,152.907
C01719=1091.947,236.078,-75.377,176.810,19.979,152.907
C01720=1091.956,236.452,-75.416,176.815,19.982,152.907
C01721=1091.965,236.826,-75.455,176.819,19.985,152.907
C01722=1091.971,237.075,-75.481,176.822,19.987,152.907
C01723=1091.976,237.324,-75.508,176.825,19.989,152.907
C01724=1091.981,237.572,-75.533,176.828,19.992,152.907
C01725=1091.987,237.820,-75.560,176.830,19.993,152.907
C01726=1091.992,238.069,-75.586,176.834,19.995,152.907
C01727=1091.999,238.317,-75.612,176.837,19.998,152.907
C01728=1092.004,238.566,-75.638,176.839,19.999,152.907
C01729=1092.010,238.815,-75.665,176.843,20.002,152.907
C01730=1092.016,239.064,-75.691,176.846,20.004,152.907
C01731=1092.021,239.312,-75.717,176.849,20.005,152.906
C01732=1092.027,239.561,-75.743,176.852,20.008,152.906
C01733=1092.033,239.809,-75.770,176.855,20.010,152.906
C01734=1092.038,240.058,-75.796,176.857,20.012,152.906
C01735=1092.044,240.307,-75.822,176.861,20.014,152.906
C01736=1092.050,240.555,-75.849,176.863,20.016,152.906
C01737=1092.055,240.804,-75.875,176.866,20.018,152.906
C01738=1092.061,241.052,-75.902,176.870,20.020,152.906
C01739=1092.067,241.301,-75.928,176.872,20.022,152.906
C01740=1092.072,241.549,-75.954,176.876,20.024,152.906
C01741=1092.077,241.797,-75.981,176.879,20.026,152.906
C01742=1092.083,242.046,-76.007,176.881,20.028,152.906
C01743=1092.089,242.295,-76.033,176.885,20.030,152.906
C01744=1092.094,242.543,-76.060,176.888,20.033,152.906
C01745=1092.100,242.791,-76.086,176.890,20.035,152.906
C01746=1092.106,243.040,-76.113,176.894,20.037,152.906
C01747=1092.112,243.289,-76.139,176.897,20.039,152.906
C01748=1092.118,243.538,-76.166,176.899,20.041,152.906
C01749=1092.122,243.786,-76.193,176.902,20.043,152.906
C01750=1092.128,244.034,-76.220,176.906,20.045,152.905
C01751=1092.133,244.283,-76.245,176.908,20.047,152.906
C01752=1092.139,244.531,-76.272,176.912,20.049,152.905
C01753=1092.145,244.780,-76.299,176.915,20.052,152.905
C01754=1092.151,245.029,-76.326,176.917,20.053,152.905
C01755=1092.156,245.278,-76.353,176.920,20.056,152.905
C01756=1092.162,245.526,-76.380,176.924,20.058,152.905
C01757=1092.168,245.774,-76.406,176.926,20.060,152.905
C01758=1092.173,246.023,-76.432,176.929,20.062,152.905
C01759=1092.178,246.272,-76.459,176.933,20.065,152.905
C01760=1092.184,246.520,-76.486,176.935,20.066,152.905
C01761=1092.190,246.769,-76.513,176.938,20.069,152.905
C01762=1092.196,247.017,-76.539,176.942,20.071,152.905
C01763=1092.201,247.266,-76.567,176.944,20.073,152.905
C01764=1092.207,247.514,-76.593,176.947,20.075,152.905
C01765=1092.212,247.762,-76.620,176.951,20.077,152.905
C01766=1092.217,248.011,-76.647,176.953,20.079,152.905
C01767=1092.223,248.259,-76.674,176.956,20.082,152.905
C01768=1092.228,248.508,-76.701,176.959,20.084,152.905
C01769=1092.234,248.756,-76.728,176.963,20.086,152.905
C01770=1092.242,249.124,-76.768,176.967,20.089,152.905
C01771=1092.251,249.491,-76.807,176.971,20.092,152.905
C01772=1092.259,249.858,-76.848,176.976,20.096,152.905
C01773=1092.267,250.225,-76.888,176.980,20.099,152.905
C01774=1092.272,250.474,-76.915,176.983,20.101,152.905
C01775=1092.278,250.722,-76.941,176.986,20.103,152.905
C01776=1092.283,250.971,-76.969,176.989,20.106,152.905
C01777=1092.289,251.219,-76.995,176.992,20.108,152.905
C01778=1092.294,251.467,-77.023,176.995,20.110,152.905
C01779=1092.301,251.716,-77.050,176.998,20.112,152.905
C01780=1092.306,251.965,-77.077,177.001,20.114,152.905
C01781=1092.312,252.213,-77.104,177.004,20.117,152.905
C01782=1092.317,252.462,-77.131,177.007,20.119,152.905
C01783=1092.323,252.710,-77.159,177.010,20.121,152.905
C01784=1092.328,252.958,-77.186,177.013,20.123,152.904
C01785=1092.334,253.207,-77.213,177.016,20.125,152.905
C01786=1092.339,253.456,-77.241,177.019,20.127,152.904
C01787=1092.345,253.704,-77.268,177.023,20.130,152.904
C01788=1092.350,253.953,-77.295,177.025,20.132,152.904
C01789=1092.356,254.200,-77.322,177.028,20.134,152.904
C01790=1092.361,254.449,-77.349,177.031,20.137,152.904
C01791=1092.368,254.698,-77.376,177.034,20.138,152.904
C01792=1092.373,254.946,-77.404,177.037,20.141,152.904
C01793=1092.378,255.195,-77.432,177.040,20.143,152.904
C01794=1092.384,255.443,-77.458,177.044,20.145,152.904
C01795=1092.390,255.692,-77.487,177.046,20.147,152.904
C01796=1092.396,255.940,-77.513,177.049,20.149,152.904
C01797=1092.401,256.188,-77.541,177.053,20.152,152.904
C01798=1092.407,256.437,-77.568,177.056,20.154,152.904
C01799=1092.413,256.685,-77.596,177.058,20.156,152.904
C01800=1092.418,256.934,-77.623,177.061,20.159,152.904
C01801=1092.424,257.182,-77.651,177.065,20.161,152.904
C01802=1092.429,257.431,-77.678,177.068,20.163,152.904
C01803=1092.436,257.679,-77.706,177.071,20.165,152.904
C01804=1092.441,257.928,-77.733,177.074,20.167,152.904
C01805=1092.446,258.176,-77.761,177.077,20.169,152.904
C01806=1092.452,258.425,-77.788,177.080,20.172,152.904
C01807=1092.458,258.673,-77.816,177.083,20.173,152.904
C01808=1092.464,258.920,-77.843,177.086,20.176,152.904
C01809=1092.469,259.170,-77.871,177.089,20.178,152.904
C01810=1092.475,259.418,-77.899,177.092,20.180,152.904
C01811=1092.481,259.667,-77.926,177.095,20.182,152.904
C01812=1092.486,259.915,-77.954,177.098,20.185,152.904
C01813=1092.492,260.163,-77.982,177.101,20.187,152.904
C01814=1092.498,260.412,-78.009,177.105,20.189,152.904
